# B&R Automation Studio project CombinedLinenSoiledA9KAN
Automation Studio 4.10.2.37

## Configuration CP1584

CPU 5APC2200.AL14-000, AutomationRuntime D4.91, Build 4.1.2, Safety 0.0, Vc V4.72.3

### Task classes (Cpu.sw)
```
Cyclic#2 (cycle 10000 us, tolerance 10000 us):
  zzstd <- Sequences.zzstd.prg
  zztc2str <- Sequences.zztc2str.prg
  zzforcei <- Sequences.zzforcei.prg
  zzconst <- Sequences.zzconst.prg
  zztrip <- Sequences.zztrip.prg
  zzbagsfl <- Sequences.zzbagsfl.prg
  zzbitcal <- Sequences.zzbitcal.prg
  zcusfifo <- Sequences.zcusfifo.prg
  zzStnSer <- Sequences.10ms.zzStnSer.prg
  1_stnsa <- Sequences.10ms.1_stnsa.prg
  2_belt1 <- Sequences.10ms.2_belt1.prg
  3_slu_1 <- Sequences.10ms.3_slu_1.prg
  4_spn1 <- Sequences.10ms.4_spn1.prg
  5_spf1 <- Sequences.10ms.5_spf1.prg
  6_sdc1 <- Sequences.10ms.6_sdc1.prg
  7_sdc2 <- Sequences.10ms.7_sdc2.prg
  8_svc1 <- Sequences.10ms.8_svc1.prg
  9_sic1 <- Sequences.10ms.9_sic1.prg
  10_bson <- Sequences.10ms.10_bson.prg
  11_bsoff <- Sequences.10ms.11_bsoff.prg
  12_svc2 <- Sequences.10ms.12_svc2.prg
  ssr_sortbe <- Sequences.10ms.ssr_sortbelt.prg
  can_live <- Sequences.can_live.prg
  zzio <- Sequences.zzio.prg
  zztcpip <- Sequences.zztcpip.prg
  zzuld_3 <- Sequences.zzuld_3.prg
  zzreport <- Sequences.zzreport.prg
  zztc2end <- Sequences.zztc2end.prg
Cyclic#4:
  Kan_Drv <- Mewa.KanLink.Kan_Drv.prg [disabled]
  mnEth <- Mewa.KGFramework.Pkg_mnEth.mnEth.prg
  BatchInfo <- Mewa.KanLink.BatchInfo.prg
  zzKanLink <- Mewa.KanLink.zzKanLink.prg [disabled]
Cyclic#5:
  zzweigh <- zzweigh.prg
  can_drv2 <- Mewa.200ms.CAN.can_drv2.prg
  zzalarms <- Sequences.zzalarms.prg
  zzstn_q <- Sequences.zzstn_q.prg
  zztime <- zztime.prg
  zztc2end1 <- zztc2end.prg
DataObjects: can_cmd <- Mewa.200ms.CAN.can_cmd.dob
Binaries: TCData, udbdef, sysconf, ashwd, asfw, arconfig, iomap, ashwac, mvLoader
Libraries: DataBackUp, mnParamLib, KanLinkLib, KGstdLib, KL_UserLib, AsDb, standard, runtime, FileIO, Ethernet, dvframe, DataObj, OPERATOR, CAN_Lib, AsTime, AsString, SupLib4, sys_lib, AsTCP, KGstring, Visapi, AsETH, AsBrStr, AsBrWStr, AsUSB, AsMem, AsArLog, AsUDP, brsystem, AsIODiag, AsARCfg, AsIecCon, IecCheck, zzSQL_Lib, arssl
```

### Hardware
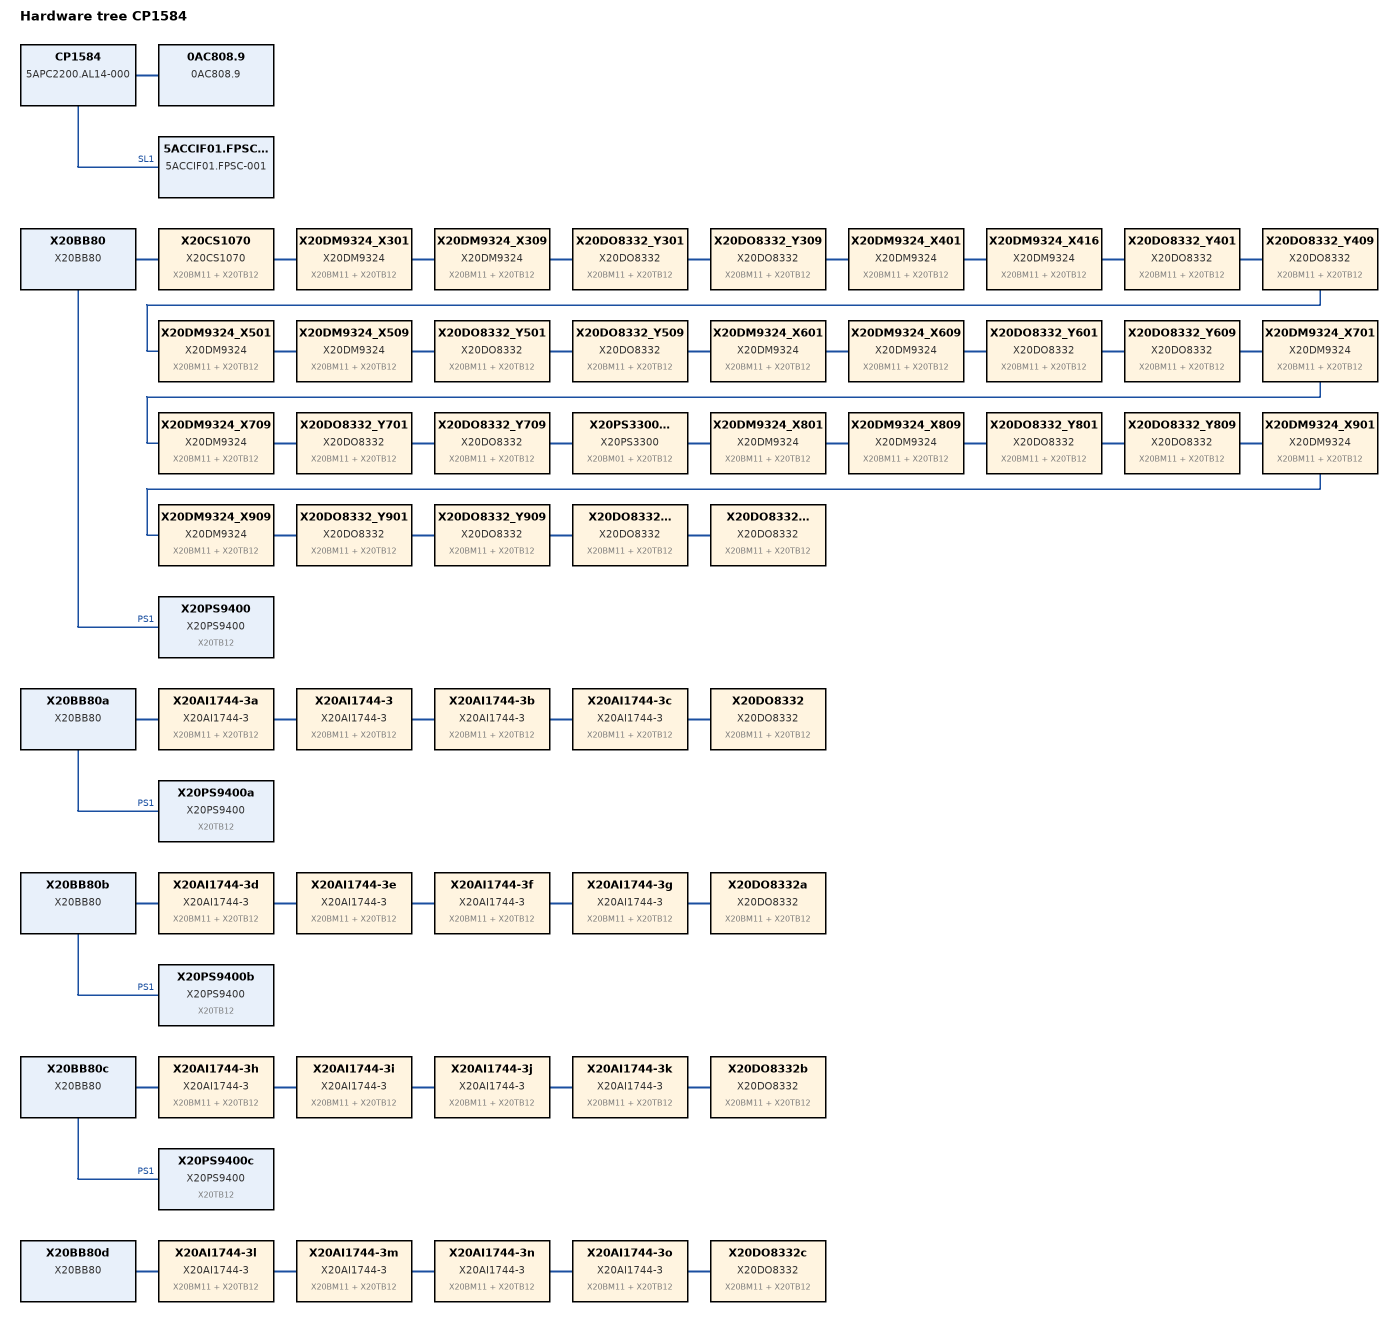
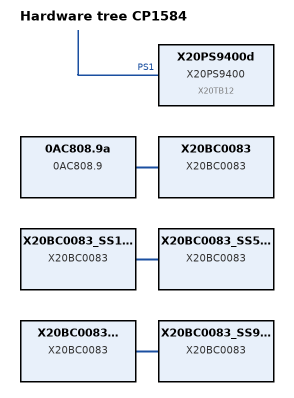
```
0AC808.9 : 0AC808.9 v1.0.0.0  [ETH1 -> CP1584.IF3 [Cable Type=PowerlinkCable, Length=10, Version=1.0.0.3]]
0AC808.9a : 0AC808.9 v1.0.0.0  [ETH2 -> X20BC0083.PLK1 [Cable Type=PowerlinkCable, Length=10, Version=1.0.0.3]; ETH4 -> X20BC0083_SS1-4.PLK2 [Cable Type=PowerlinkCable, Length=10, Version=1.0.0.3]]
5ACCIF01.FPSC-001 : 5ACCIF01.FPSC-001 v1.9.1.0  [SL -> CP1584.SL1]
  Connector IF1:
    DNAConfiguration = manual
CP1584 : 5APC2200.AL14-000 v2.0.3.0
  Connector IF3:
    AssignedOperatingSystem = ARemb
    ActivateDevice = 1
    Baudrate = 100
    InaNodeNumber = 21
    ActivateANSL = 0
  Connector IF4:
    AssignedOperatingSystem = ARemb
    ActivateDevice = 1
    Mode = Manual
    InternetAddress = 10.8.4.20
    SubnetMask = 255.255.240.0
  Connector IF5:
    AssignedOperatingSystem = ARemb
  Connector IF6:
    AssignedOperatingSystem = ARemb
  ConfigurationID = AS4_2_BaseStandard_Supertrack
  UserPartitionSize = 0
  UserRamDevice = PCI.1.PPC21xx.SRAM
  UserRamSize = 200000
  RemMemDevice = PCI.1.PPC21xx.SRAM
  RemMemSize = 200000
  PermanentPvSize = 46756
  RemanentGlobalPvSize = 8944
  VolatileGlobalPvSize = 450000
  EnableUsbRemoteInstall = 1
  EnableCfRemoteInstall = 1
  Cyclic1Duration = 1000
  Cyclic1Tolerance = 1000
  Cyclic2Duration = 10000
  Cyclic2Tolerance = 10000
  FileDevice1
  FileDeviceName1 = USBStick
  FileDevicePath1 = /bd0\
  FileDevice2
  FileDeviceName2 = UserPart
  FileDevicePath2 = F:\
  EthernetHostName = SupertrackPLC
  EthernetDefaultGateway = 10.8.15.254
  FtpUser1
  FtpUsername1 = admin
  FtpUserPassword1 = vwQCGOhDKwuFhUdMhisKVJgiKzmoNTQazzJQnTTJsZU=  // admin
  FtpUserSalt1 = XFuy8Eo/
  FTPAccessRight1 = 0
  ActivateOpcUa = 1
  OpcUaInformationModels_PV_Version = 1
X20AI1744-3 : X20AI1744-3 v1.7.0.0  [SS1 -> X20TB12ai.SS; SL -> X20BM11af.SL1]
  Supervision = off
X20AI1744-3a : X20AI1744-3 v1.7.0.0  [SS1 -> X20TB12ah.SS; SL -> X20BM11ae.SL1]
  Supervision = off
X20AI1744-3b : X20AI1744-3 v1.7.0.0  [SS1 -> X20TB12aj.SS; SL -> X20BM11ag.SL1]
  Supervision = off
X20AI1744-3c : X20AI1744-3 v1.7.0.0  [SS1 -> X20TB12ak.SS; SL -> X20BM11ah.SL1]
  Supervision = off
X20AI1744-3d : X20AI1744-3 v1.7.0.0  [SS1 -> X20TB12ap.SS; SL -> X20BM11aj.SL1]
  Supervision = off
X20AI1744-3e : X20AI1744-3 v1.7.0.0  [SS1 -> X20TB12aq.SS; SL -> X20BM11ak.SL1]
  Supervision = off
X20AI1744-3f : X20AI1744-3 v1.7.0.0  [SS1 -> X20TB12ar.SS; SL -> X20BM11al.SL1]
  Supervision = off
X20AI1744-3g : X20AI1744-3 v1.7.0.0  [SS1 -> X20TB12as.SS; SL -> X20BM11am.SL1]
  Supervision = off
X20AI1744-3h : X20AI1744-3 v1.7.0.0  [SS1 -> X20TB12au.SS; SL -> X20BM11ao.SL1]
  Supervision = off
X20AI1744-3i : X20AI1744-3 v1.7.0.0  [SS1 -> X20TB12av.SS; SL -> X20BM11ap.SL1]
  Supervision = off
X20AI1744-3j : X20AI1744-3 v1.7.0.0  [SS1 -> X20TB12aw.SS; SL -> X20BM11aq.SL1]
  Supervision = off
X20AI1744-3k : X20AI1744-3 v1.7.0.0  [SS1 -> X20TB12ax.SS; SL -> X20BM11ar.SL1]
  Supervision = off
X20AI1744-3l : X20AI1744-3 v1.7.0.0  [SS1 -> X20TB12az.SS; SL -> X20BM11at.SL1]
  Supervision = off
X20AI1744-3m : X20AI1744-3 v1.7.0.0  [SS1 -> X20TB12ba.SS; SL -> X20BM11au.SL1]
  Supervision = off
X20AI1744-3n : X20AI1744-3 v1.7.0.0  [SS1 -> X20TB12bb.SS; SL -> X20BM11av.SL1]
  Supervision = off
X20AI1744-3o : X20AI1744-3 v1.7.0.0  [SS1 -> X20TB12bc.SS; SL -> X20BM11aw.SL1]
  Supervision = off
X20BB80 : X20BB80 v1.1.0.0
X20BB80a : X20BB80 v1.1.0.0
X20BB80b : X20BB80 v1.1.0.0
X20BB80c : X20BB80 v1.1.0.0
X20BB80d : X20BB80 v1.1.0.0
X20BC0083 : X20BC0083 v2.14.0.0  [PLK1 -> 0AC808.9a.ETH2 [Cable Type=PowerlinkCable, Length=10, Version=1.0.0.3]; PLK2 -> 5ACCIF01.FPSC-001.IF1 [Cable Type=PowerlinkCable, Length=10, Version=1.0.0.3]; SL -> X20BB80.SL1]
  Supervision = off
X20BC0083_SS1-4 : X20BC0083 v2.14.0.0  [PLK1 -> X20BC0083_SS5-8.PLK1 [Cable Type=PowerlinkCable, Length=10, Version=1.0.0.3]; PLK2 -> 0AC808.9a.ETH4 [Cable Type=PowerlinkCable, Length=10, Version=1.0.0.3]; SL -> X20BB80a.SL1]
  Supervision = off
X20BC0083_SS13-16 : X20BC0083 v2.14.0.0  [PLK2 -> X20BC0083_SS9-12.PLK1 (NodeNumber=5) [Cable Type=PowerlinkCable, Length=10, Version=1.0.0.3]; SL -> X20BB80d.SL1]
  Supervision = off
X20BC0083_SS5-8 : X20BC0083 v2.14.0.0  [PLK1 -> X20BC0083_SS1-4.PLK1 (NodeNumber=3) [Cable Type=PowerlinkCable, Length=10, Version=1.0.0.3]; PLK2 -> X20BC0083_SS9-12.PLK2 (NodeNumber=3) [Cable Type=PowerlinkCable, Length=10, Version=1.0.0.3]; SL -> X20BB80b.SL1]
  Supervision = off
X20BC0083_SS9-12 : X20BC0083 v2.14.0.0  [PLK1 -> X20BC0083_SS13-16.PLK2 (NodeNumber=4) [Cable Type=PowerlinkCable, Length=10, Version=1.0.0.3]; PLK2 -> X20BC0083_SS5-8.PLK2 (NodeNumber=4) [Cable Type=PowerlinkCable, Length=10, Version=1.0.0.3]; SL -> X20BB80c.SL1]
  Supervision = off
X20BM01 : X20BM01 v2.1.0.0  [X2X1 -> X20BM11t.X2X2]
X20BM11 : X20BM11 v1.1.0.0  [X2X1 -> X20BB80.IF1]
X20BM11a : X20BM11 v1.1.0.0  [X2X1 -> X20BM11.X2X2]
X20BM11aa : X20BM11 v1.1.0.0  [X2X1 -> X20BM11z.X2X2]
X20BM11ab : X20BM11 v1.1.0.0  [X2X1 -> X20BM11aa.X2X2]
X20BM11ac : X20BM11 v1.1.0.0  [X2X1 -> X20BM11ab.X2X2]
X20BM11ad : X20BM11 v1.1.0.0  [X2X1 -> X20BM11ac.X2X2]
X20BM11ae : X20BM11 v1.1.0.0  [X2X1 -> X20BB80a.IF1]
X20BM11af : X20BM11 v1.1.0.0  [X2X1 -> X20BM11ae.X2X2]
X20BM11ag : X20BM11 v1.1.0.0  [X2X1 -> X20BM11af.X2X2]
X20BM11ah : X20BM11 v1.1.0.0  [X2X1 -> X20BM11ag.X2X2]
X20BM11ai : X20BM11 v1.1.0.0  [X2X1 -> X20BM11ah.X2X2]
X20BM11aj : X20BM11 v1.1.0.0  [X2X1 -> X20BB80b.IF1]
X20BM11ak : X20BM11 v1.1.0.0  [X2X1 -> X20BM11aj.X2X2]
X20BM11al : X20BM11 v1.1.0.0  [X2X1 -> X20BM11ak.X2X2]
X20BM11am : X20BM11 v1.1.0.0  [X2X1 -> X20BM11al.X2X2]
X20BM11an : X20BM11 v1.1.0.0  [X2X1 -> X20BM11am.X2X2]
X20BM11ao : X20BM11 v1.1.0.0  [X2X1 -> X20BB80c.IF1]
X20BM11ap : X20BM11 v1.1.0.0  [X2X1 -> X20BM11ao.X2X2]
X20BM11aq : X20BM11 v1.1.0.0  [X2X1 -> X20BM11ap.X2X2]
X20BM11ar : X20BM11 v1.1.0.0  [X2X1 -> X20BM11aq.X2X2]
X20BM11as : X20BM11 v1.1.0.0  [X2X1 -> X20BM11ar.X2X2]
X20BM11at : X20BM11 v1.1.0.0  [X2X1 -> X20BB80d.IF1]
X20BM11au : X20BM11 v1.1.0.0  [X2X1 -> X20BM11at.X2X2]
X20BM11av : X20BM11 v1.1.0.0  [X2X1 -> X20BM11au.X2X2]
X20BM11aw : X20BM11 v1.1.0.0  [X2X1 -> X20BM11av.X2X2]
X20BM11ax : X20BM11 v1.1.0.0  [X2X1 -> X20BM11aw.X2X2]
X20BM11b : X20BM11 v1.1.0.0  [X2X1 -> X20BM11a.X2X2]
X20BM11c : X20BM11 v1.1.0.0  [X2X1 -> X20BM11b.X2X2]
X20BM11d : X20BM11 v1.1.0.0  [X2X1 -> X20BM11e.X2X2]
X20BM11e : X20BM11 v1.1.0.0  [X2X1 -> X20BM11c.X2X2]
X20BM11f : X20BM11 v1.1.0.0  [X2X1 -> X20BM11d.X2X2]
X20BM11g : X20BM11 v1.1.0.0  [X2X1 -> X20BM11s.X2X2]
X20BM11h : X20BM11 v1.1.0.0  [X2X1 -> X20BM11f.X2X2]
X20BM11i : X20BM11 v1.1.0.0  [X2X1 -> X20BM11h.X2X2]
X20BM11j : X20BM11 v1.1.0.0  [X2X1 -> X20BM11i.X2X2]
X20BM11k : X20BM11 v1.1.0.0  [X2X1 -> X20BM11j.X2X2]
X20BM11l : X20BM11 v1.1.0.0  [X2X1 -> X20BM11k.X2X2]
X20BM11m : X20BM11 v1.1.0.0  [X2X1 -> X20BM11l.X2X2]
X20BM11n : X20BM11 v1.1.0.0  [X2X1 -> X20BM11m.X2X2]
X20BM11o : X20BM11 v1.1.0.0  [X2X1 -> X20BM11n.X2X2]
X20BM11p : X20BM11 v1.1.0.0  [X2X1 -> X20BM11o.X2X2]
X20BM11q : X20BM11 v1.1.0.0  [X2X1 -> X20BM11p.X2X2]
X20BM11r : X20BM11 v1.1.0.0  [X2X1 -> X20BM11q.X2X2]
X20BM11s : X20BM11 v1.1.0.0  [X2X1 -> X20BM11r.X2X2]
X20BM11t : X20BM11 v1.1.0.0  [X2X1 -> X20BM11g.X2X2]
X20BM11u : X20BM11 v1.1.0.0  [X2X1 -> X20BM01.X2X2]
X20BM11v : X20BM11 v1.1.0.0  [X2X1 -> X20BM11u.X2X2]
X20BM11w : X20BM11 v1.1.0.0  [X2X1 -> X20BM11v.X2X2]
X20BM11x : X20BM11 v1.1.0.0  [X2X1 -> X20BM11w.X2X2]
X20BM11y : X20BM11 v1.1.0.0  [X2X1 -> X20BM11x.X2X2]
X20BM11z : X20BM11 v1.1.0.0  [X2X1 -> X20BM11y.X2X2]
X20CS1070 : X20CS1070 v1.8.0.0  [SS1 -> X20TB12af.SS; SL -> X20BM11.SL1]
  Connector IF1:
    Baudrate = 250000
  FunctionModel = Stream1xCan
  Supervision = off
X20DM9324_X301 : X20DM9324 v1.2.0.0  [SS1 -> X20TB12a.SS; SL -> X20BM11a.SL1]
  Supervision = off
X20DM9324_X309 : X20DM9324 v1.2.0.0  [SS1 -> X20TB12b.SS; SL -> X20BM11b.SL1]
  Supervision = off
X20DM9324_X401 : X20DM9324 v1.2.0.0  [SS1 -> X20TB12d.SS; SL -> X20BM11d.SL1]
  Supervision = off
X20DM9324_X416 : X20DM9324 v1.2.0.0  [SS1 -> X20TB12f.SS; SL -> X20BM11f.SL1]
  Supervision = off
X20DM9324_X501 : X20DM9324 v1.2.0.0  [SS1 -> X20TB12j.SS; SL -> X20BM11j.SL1]
  Supervision = off
X20DM9324_X509 : X20DM9324 v1.2.0.0  [SS1 -> X20TB12k.SS; SL -> X20BM11k.SL1]
  Supervision = off
X20DM9324_X601 : X20DM9324 v1.2.0.0  [SS1 -> X20TB12n.SS; SL -> X20BM11n.SL1]
  Supervision = off
X20DM9324_X609 : X20DM9324 v1.2.0.0  [SS1 -> X20TB12o.SS; SL -> X20BM11o.SL1]
  Supervision = off
X20DM9324_X701 : X20DM9324 v1.2.0.0  [SS1 -> X20TB12r.SS; SL -> X20BM11r.SL1]
  Supervision = off
X20DM9324_X709 : X20DM9324 v1.2.0.0  [SS1 -> X20TB12s.SS; SL -> X20BM11s.SL1]
  Supervision = off
X20DM9324_X801 : X20DM9324 v1.2.0.0  [SS1 -> X20TB12u.SS; SL -> X20BM11u.SL1]
  Supervision = off
X20DM9324_X809 : X20DM9324 v1.2.0.0  [SS1 -> X20TB12v.SS; SL -> X20BM11v.SL1]
  Supervision = off
X20DM9324_X901 : X20DM9324 v1.2.0.0  [SS1 -> X20TB12z.SS; SL -> X20BM11y.SL1]
  Supervision = off
X20DM9324_X909 : X20DM9324 v1.2.0.0  [SS1 -> X20TB12aa.SS; SL -> X20BM11z.SL1]
  Supervision = off
X20DO8332 : X20DO8332 v1.5.0.0  [SS1 -> X20TB12al.SS; SL -> X20BM11ai.SL1]
  Supervision = off
X20DO8332_Y1001 : X20DO8332 v1.5.0.0  [SS1 -> X20TB12ad.SS; SL -> X20BM11ac.SL1]
  Supervision = off
X20DO8332_Y1009 : X20DO8332 v1.5.0.0  [SS1 -> X20TB12ae.SS; SL -> X20BM11ad.SL1]
  Supervision = off
X20DO8332_Y301 : X20DO8332 v1.5.0.0  [SS1 -> X20TB12c.SS; SL -> X20BM11c.SL1]
  Supervision = off
X20DO8332_Y309 : X20DO8332 v1.5.0.0  [SS1 -> X20TB12e.SS; SL -> X20BM11e.SL1]
  Supervision = off
X20DO8332_Y401 : X20DO8332 v1.5.0.0  [SS1 -> X20TB12h.SS; SL -> X20BM11h.SL1]
  Supervision = off
X20DO8332_Y409 : X20DO8332 v1.5.0.0  [SS1 -> X20TB12i.SS; SL -> X20BM11i.SL1]
  Supervision = off
X20DO8332_Y501 : X20DO8332 v1.5.0.0  [SS1 -> X20TB12l.SS; SL -> X20BM11l.SL1]
  Supervision = off
X20DO8332_Y509 : X20DO8332 v1.5.0.0  [SS1 -> X20TB12m.SS; SL -> X20BM11m.SL1]
  Supervision = off
X20DO8332_Y601 : X20DO8332 v1.5.0.0  [SS1 -> X20TB12p.SS; SL -> X20BM11p.SL1]
  Supervision = off
X20DO8332_Y609 : X20DO8332 v1.5.0.0  [SS1 -> X20TB12q.SS; SL -> X20BM11q.SL1]
  Supervision = off
X20DO8332_Y701 : X20DO8332 v1.5.0.0  [SS1 -> X20TB12g.SS; SL -> X20BM11g.SL1]
  Supervision = off
X20DO8332_Y709 : X20DO8332 v1.5.0.0  [SS1 -> X20TB12t.SS; SL -> X20BM11t.SL1]
  Supervision = off
X20DO8332_Y801 : X20DO8332 v1.5.0.0  [SS1 -> X20TB12x.SS; SL -> X20BM11w.SL1]
  Supervision = off
X20DO8332_Y809 : X20DO8332 v1.5.0.0  [SS1 -> X20TB12y.SS; SL -> X20BM11x.SL1]
  Supervision = off
X20DO8332_Y901 : X20DO8332 v1.5.0.0  [SS1 -> X20TB12ab.SS; SL -> X20BM11aa.SL1]
  Supervision = off
X20DO8332_Y909 : X20DO8332 v1.5.0.0  [SS1 -> X20TB12ac.SS; SL -> X20BM11ab.SL1]
  Supervision = off
X20DO8332a : X20DO8332 v1.5.0.0  [SS1 -> X20TB12at.SS; SL -> X20BM11an.SL1]
  Supervision = off
X20DO8332b : X20DO8332 v1.5.0.0  [SS1 -> X20TB12ay.SS; SL -> X20BM11as.SL1]
  Supervision = off
X20DO8332c : X20DO8332 v1.5.0.0  [SS1 -> X20TB12bd.SS; SL -> X20BM11ax.SL1]
  Supervision = off
X20PS3300_Power : X20PS3300 v1.3.0.0  [SS1 -> X20TB12w.SS; SL -> X20BM01.SL1]
  Supervision = off
X20PS9400 : X20PS9400 v1.8.0.0  [SS1 -> X20TB12.SS; PS -> X20BB80.PS1]
  Supervision = off
X20PS9400a : X20PS9400 v1.8.0.0  [SS1 -> X20TB12ag.SS; PS -> X20BB80a.PS1]
  Supervision = off
X20PS9400b : X20PS9400 v1.8.0.0  [SS1 -> X20TB12am.SS; PS -> X20BB80b.PS1]
  Supervision = off
X20PS9400c : X20PS9400 v1.8.0.0  [SS1 -> X20TB12an.SS; PS -> X20BB80c.PS1]
  Supervision = off
X20PS9400d : X20PS9400 v1.8.0.0  [SS1 -> X20TB12ao.SS; PS -> X20BB80d.PS1]
  Supervision = off
X20TB12 : X20TB12 v1.0.0.0
X20TB12a : X20TB12 v1.0.0.0
X20TB12aa : X20TB12 v1.0.0.0
X20TB12ab : X20TB12 v1.0.0.0
X20TB12ac : X20TB12 v1.0.0.0
X20TB12ad : X20TB12 v1.0.0.0
X20TB12ae : X20TB12 v1.0.0.0
X20TB12af : X20TB12 v1.0.0.0
X20TB12ag : X20TB12 v1.0.0.0
X20TB12ah : X20TB12 v1.0.0.0
X20TB12ai : X20TB12 v1.0.0.0
X20TB12aj : X20TB12 v1.0.0.0
X20TB12ak : X20TB12 v1.0.0.0
X20TB12al : X20TB12 v1.0.0.0
X20TB12am : X20TB12 v1.0.0.0
X20TB12an : X20TB12 v1.0.0.0
X20TB12ao : X20TB12 v1.0.0.0
X20TB12ap : X20TB12 v1.0.0.0
X20TB12aq : X20TB12 v1.0.0.0
X20TB12ar : X20TB12 v1.0.0.0
X20TB12as : X20TB12 v1.0.0.0
X20TB12at : X20TB12 v1.0.0.0
X20TB12au : X20TB12 v1.0.0.0
X20TB12av : X20TB12 v1.0.0.0
X20TB12aw : X20TB12 v1.0.0.0
X20TB12ax : X20TB12 v1.0.0.0
X20TB12ay : X20TB12 v1.0.0.0
X20TB12az : X20TB12 v1.0.0.0
X20TB12b : X20TB12 v1.0.0.0
X20TB12ba : X20TB12 v1.0.0.0
X20TB12bb : X20TB12 v1.0.0.0
X20TB12bc : X20TB12 v1.0.0.0
X20TB12bd : X20TB12 v1.0.0.0
X20TB12c : X20TB12 v1.0.0.0
X20TB12d : X20TB12 v1.0.0.0
X20TB12e : X20TB12 v1.0.0.0
X20TB12f : X20TB12 v1.0.0.0
X20TB12g : X20TB12 v1.0.0.0
X20TB12h : X20TB12 v1.0.0.0
X20TB12i : X20TB12 v1.0.0.0
X20TB12j : X20TB12 v1.0.0.0
X20TB12k : X20TB12 v1.0.0.0
X20TB12l : X20TB12 v1.0.0.0
X20TB12m : X20TB12 v1.0.0.0
X20TB12n : X20TB12 v1.0.0.0
X20TB12o : X20TB12 v1.0.0.0
X20TB12p : X20TB12 v1.0.0.0
X20TB12q : X20TB12 v1.0.0.0
X20TB12r : X20TB12 v1.0.0.0
X20TB12s : X20TB12 v1.0.0.0
X20TB12t : X20TB12 v1.0.0.0
X20TB12u : X20TB12 v1.0.0.0
X20TB12v : X20TB12 v1.0.0.0
X20TB12w : X20TB12 v1.0.0.0
X20TB12x : X20TB12 v1.0.0.0
X20TB12y : X20TB12 v1.0.0.0
X20TB12z : X20TB12 v1.0.0.0
```

### Cpu.per - CP1584/Cpu.per
```iecst
(********************************************************************
 * COPYRIGHT -- HP
 ********************************************************************
 * File: Cpu.per
 * Author: treamsbottom
 * Created: March 03, 2014
 ********************************************************************
 * Declaration of permanent variables
 ********************************************************************)
VAR_CONFIG
	Bag AT %M0; (* *)
	C AT %MW16000; (* *)
	D AT %MW16200; (* *)
	(*D32 AT %MD32200; (* *)
	ReportBuffer AT %M36200; (* *)
	SQL AT %M44200; (* *)
END_VAR
```

### IoMap.iom - CP1584/IoMap.iom
```iecst
(********************************************************************
 * COPYRIGHT --
 ********************************************************************
 * File: IoMap.iom
 * Author: Dave
 * Created: November 19, 2010
 ********************************************************************
 * IO mapping file
 ********************************************************************)
VAR_CONFIG
	X[3].X01 AT %QX."X20DO8332_Y301".DigitalOutput01;
	X[3].X02 AT %QX."X20DO8332_Y301".DigitalOutput02;
	X[3].X03 AT %QX."X20DO8332_Y301".DigitalOutput03;
	X[3].X04 AT %QX."X20DO8332_Y301".DigitalOutput04;
	X[3].X05 AT %QX."X20DO8332_Y301".DigitalOutput05;
	X[3].X06 AT %QX."X20DO8332_Y301".DigitalOutput06;
	X[3].X07 AT %QX."X20DO8332_Y301".DigitalOutput07;
	X[3].X08 AT %QX."X20DO8332_Y301".DigitalOutput08;
	X[3].X09 AT %IX."X20DM9324_X309".DigitalInput01;
	X[3].X10 AT %IX."X20DM9324_X309".DigitalInput02;
	X[3].X11 AT %IX."X20DM9324_X309".DigitalInput03;
	X[3].X12 AT %IX."X20DM9324_X309".DigitalInput04;
	X[3].X13 AT %IX."X20DM9324_X309".DigitalInput05;
	X[3].X14 AT %IX."X20DM9324_X309".DigitalInput06;
	X[3].X15 AT %IX."X20DM9324_X309".DigitalInput07;
	X[3].X16 AT %IX."X20DM9324_X309".DigitalInput08;
	Y[3].Y01 AT %IX."X20DM9324_X301".DigitalInput01;
	Y[3].Y02 AT %IX."X20DM9324_X301".DigitalInput02;
	Y[3].Y03 AT %IX."X20DM9324_X301".DigitalInput03;
	Y[3].Y04 AT %IX."X20DM9324_X301".DigitalInput04;
	Y[3].Y05 AT %IX."X20DM9324_X301".DigitalInput05;
	Y[3].Y06 AT %IX."X20DM9324_X301".DigitalInput06;
	Y[3].Y07 AT %IX."X20DM9324_X301".DigitalInput07;
	Y[3].Y08 AT %IX."X20DM9324_X301".DigitalInput08;
	Y[3].Y09 AT %QX."X20DO8332_Y309".DigitalOutput01;
	Y[3].Y10 AT %QX."X20DO8332_Y309".DigitalOutput02;
	Y[3].Y11 AT %QX."X20DO8332_Y309".DigitalOutput03;
	Y[3].Y12 AT %QX."X20DO8332_Y309".DigitalOutput04;
	Y[3].Y13 AT %QX."X20DO8332_Y309".DigitalOutput05;
	Y[3].Y14 AT %QX."X20DO8332_Y309".DigitalOutput06;
	Y[3].Y15 AT %QX."X20DO8332_Y309".DigitalOutput07;
	Y[3].Y16 AT %QX."X20DO8332_Y309".DigitalOutput08;
	X[4].X01 AT %IX."X20DM9324_X401".DigitalInput01;
	X[4].X02 AT %IX."X20DM9324_X401".DigitalInput02;
	X[4].X03 AT %IX."X20DM9324_X401".DigitalInput03;
	X[4].X04 AT %IX."X20DM9324_X401".DigitalInput04;
	X[4].X05 AT %IX."X20DM9324_X401".DigitalInput05;
	X[4].X06 AT %IX."X20DM9324_X401".DigitalInput06;
	X[4].X07 AT %IX."X20DM9324_X401".DigitalInput07;
	X[4].X08 AT %IX."X20DM9324_X401".DigitalInput08;
	X[4].X09 AT %IX."X20DM9324_X416".DigitalInput01;
	X[4].X10 AT %IX."X20DM9324_X416".DigitalInput02;
	X[4].X11 AT %IX."X20DM9324_X416".DigitalInput03;
	X[4].X12 AT %IX."X20DM9324_X416".DigitalInput04;
	X[4].X13 AT %IX."X20DM9324_X416".DigitalInput05;
	X[4].X14 AT %IX."X20DM9324_X416".DigitalInput06;
	X[4].X15 AT %IX."X20DM9324_X416".DigitalInput07;
	X[4].X16 AT %IX."X20DM9324_X416".DigitalInput08;
	Y[4].Y01 AT %QX."X20DO8332_Y401".DigitalOutput01;
	Y[4].Y02 AT %QX."X20DO8332_Y401".DigitalOutput02;
	Y[4].Y03 AT %QX."X20DO8332_Y401".DigitalOutput03;
	Y[4].Y04 AT %QX."X20DO8332_Y401".DigitalOutput04;
	Y[4].Y05 AT %QX."X20DO8332_Y401".DigitalOutput05;
	Y[4].Y06 AT %QX."X20DO8332_Y401".DigitalOutput06;
	Y[4].Y07 AT %QX."X20DO8332_Y401".DigitalOutput07;
	Y[4].Y08 AT %QX."X20DO8332_Y401".DigitalOutput08;
	Y[4].Y09 AT %QX."X20DO8332_Y409".DigitalOutput01;
	Y[4].Y10 AT %QX."X20DO8332_Y409".DigitalOutput02;
	Y[4].Y11 AT %QX."X20DO8332_Y409".DigitalOutput03;
	Y[4].Y12 AT %QX."X20DO8332_Y409".DigitalOutput04;
	Y[4].Y13 AT %QX."X20DO8332_Y409".DigitalOutput05;
	Y[4].Y14 AT %QX."X20DO8332_Y409".DigitalOutput06;
	Y[4].Y15 AT %QX."X20DO8332_Y409".DigitalOutput07;
	Y[4].Y16 AT %QX."X20DO8332_Y409".DigitalOutput08;
	X[5].X01 AT %IX."X20DM9324_X501".DigitalInput01;
	X[5].X02 AT %IX."X20DM9324_X501".DigitalInput02;
	X[5].X03 AT %IX."X20DM9324_X501".DigitalInput03;
	X[5].X04 AT %IX."X20DM9324_X501".DigitalInput04;
	X[5].X05 AT %IX."X20DM9324_X501".DigitalInput05;
	X[5].X06 AT %IX."X20DM9324_X501".DigitalInput06;
	X[5].X07 AT %IX."X20DM9324_X501".DigitalInput07;
	X[5].X08 AT %IX."X20DM9324_X501".DigitalInput08;
	X[5].X09 AT %IX."X20DM9324_X509".DigitalInput01;
	X[5].X10 AT %IX."X20DM9324_X509".DigitalInput02;
	X[5].X11 AT %IX."X20DM9324_X509".DigitalInput03;
	X[5].X12 AT %IX."X20DM9324_X509".DigitalInput04;
	X[5].X13 AT %IX."X20DM9324_X509".DigitalInput05;
	X[5].X14 AT %IX."X20DM9324_X509".DigitalInput06;
	X[5].X15 AT %IX."X20DM9324_X509".DigitalInput07;
	X[5].X16 AT %IX."X20DM9324_X509".DigitalInput08;
	Y[5].Y01 AT %QX."X20DO8332_Y501".DigitalOutput01;
	Y[5].Y02 AT %QX."X20DO8332_Y501".DigitalOutput02;
	Y[5].Y03 AT %QX."X20DO8332_Y501".DigitalOutput03;
	Y[5].Y04 AT %QX."X20DO8332_Y501".DigitalOutput04;
	Y[5].Y05 AT %QX."X20DO8332_Y501".DigitalOutput05;
	Y[5].Y06 AT %QX."X20DO8332_Y501".DigitalOutput06;
	Y[5].Y07 AT %QX."X20DO8332_Y501".DigitalOutput07;
	Y[5].Y08 AT %QX."X20DO8332_Y501".DigitalOutput08;
	Y[5].Y09 AT %QX."X20DO8332_Y509".DigitalOutput01;
	Y[5].Y10 AT %QX."X20DO8332_Y509".DigitalOutput02;
	Y[5].Y11 AT %QX."X20DO8332_Y509".DigitalOutput03;
	Y[5].Y12 AT %QX."X20DO8332_Y509".DigitalOutput04;
	Y[5].Y13 AT %QX."X20DO8332_Y509".DigitalOutput05;
	Y[5].Y14 AT %QX."X20DO8332_Y509".DigitalOutput06;
	Y[5].Y15 AT %QX."X20DO8332_Y509".DigitalOutput07;
	Y[5].Y16 AT %QX."X20DO8332_Y509".DigitalOutput08;
	X[6].X01 AT %IX."X20DM9324_X601".DigitalInput01;
	X[6].X02 AT %IX."X20DM9324_X601".DigitalInput02;
	X[6].X03 AT %IX."X20DM9324_X601".DigitalInput03;
	X[6].X04 AT %IX."X20DM9324_X601".DigitalInput04;
	X[6].X05 AT %IX."X20DM9324_X601".DigitalInput05;
	X[6].X06 AT %IX."X20DM9324_X601".DigitalInput06;
	X[6].X07 AT %IX."X20DM9324_X601".DigitalInput07;
	X[6].X08 AT %IX."X20DM9324_X601".DigitalInput08;
	X[6].X09 AT %IX."X20DM9324_X609".DigitalInput01;
	X[6].X10 AT %IX."X20DM9324_X609".DigitalInput02;
	X[6].X11 AT %IX."X20DM9324_X609".DigitalInput03;
	X[6].X12 AT %IX."X20DM9324_X609".DigitalInput04;
	X[6].X13 AT %IX."X20DM9324_X609".DigitalInput05;
	X[6].X14 AT %IX."X20DM9324_X609".DigitalInput06;
	X[6].X15 AT %IX."X20DM9324_X609".DigitalInput07;
	X[6].X16 AT %IX."X20DM9324_X609".DigitalInput08;
	Y[6].Y01 AT %QX."X20DO8332_Y601".DigitalOutput01;
	Y[6].Y02 AT %QX."X20DO8332_Y601".DigitalOutput02;
	Y[6].Y03 AT %QX."X20DO8332_Y601".DigitalOutput03;
	Y[6].Y04 AT %QX."X20DO8332_Y601".DigitalOutput04;
	Y[6].Y05 AT %QX."X20DO8332_Y601".DigitalOutput05;
	Y[6].Y06 AT %QX."X20DO8332_Y601".DigitalOutput06;
	Y[6].Y07 AT %QX."X20DO8332_Y601".DigitalOutput07;
	Y[6].Y08 AT %QX."X20DO8332_Y601".DigitalOutput08;
	Y[6].Y09 AT %QX."X20DO8332_Y609".DigitalOutput01;
	Y[6].Y10 AT %QX."X20DO8332_Y609".DigitalOutput02;
	Y[6].Y11 AT %QX."X20DO8332_Y609".DigitalOutput03;
	Y[6].Y12 AT %QX."X20DO8332_Y609".DigitalOutput04;
	Y[6].Y13 AT %QX."X20DO8332_Y609".DigitalOutput05;
	Y[6].Y14 AT %QX."X20DO8332_Y609".DigitalOutput06;
	Y[6].Y15 AT %QX."X20DO8332_Y609".DigitalOutput07;
	Y[6].Y16 AT %QX."X20DO8332_Y609".DigitalOutput08;
	X[7].X01 AT %IX."X20DM9324_X701".DigitalInput01;
	X[7].X02 AT %IX."X20DM9324_X701".DigitalInput02;
	X[7].X03 AT %IX."X20DM9324_X701".DigitalInput03;
	X[7].X04 AT %IX."X20DM9324_X701".DigitalInput04;
	X[7].X05 AT %IX."X20DM9324_X701".DigitalInput05;
	X[7].X06 AT %IX."X20DM9324_X701".DigitalInput06;
	X[7].X07 AT %IX."X20DM9324_X701".DigitalInput07;
	X[7].X08 AT %IX."X20DM9324_X701".DigitalInput08;
	X[7].X09 AT %IX."X20DM9324_X709".DigitalInput01;
	X[7].X10 AT %IX."X20DM9324_X709".DigitalInput02;
	X[7].X11 AT %IX."X20DM9324_X709".DigitalInput03;
	X[7].X12 AT %IX."X20DM9324_X709".DigitalInput04;
	X[7].X13 AT %IX."X20DM9324_X709".DigitalInput05;
	X[7].X14 AT %IX."X20DM9324_X709".DigitalInput06;
	X[7].X15 AT %IX."X20DM9324_X709".DigitalInput07;
	X[7].X16 AT %IX."X20DM9324_X709".DigitalInput08;
	Y[7].Y01 AT %QX."X20DO8332_Y701".DigitalOutput01;
	Y[7].Y02 AT %QX."X20DO8332_Y701".DigitalOutput02;
	Y[7].Y03 AT %QX."X20DO8332_Y701".DigitalOutput03;
	Y[7].Y04 AT %QX."X20DO8332_Y701".DigitalOutput04;
	Y[7].Y05 AT %QX."X20DO8332_Y701".DigitalOutput05;
	Y[7].Y06 AT %QX."X20DO8332_Y701".DigitalOutput06;
	Y[7].Y07 AT %QX."X20DO8332_Y701".DigitalOutput07;
	Y[7].Y08 AT %QX."X20DO8332_Y701".DigitalOutput08;
	Y[7].Y09 AT %QX."X20DO8332_Y709".DigitalOutput01;
	Y[7].Y10 AT %QX."X20DO8332_Y709".DigitalOutput02;
	Y[7].Y11 AT %QX."X20DO8332_Y709".DigitalOutput03;
	Y[7].Y12 AT %QX."X20DO8332_Y709".DigitalOutput04;
	Y[7].Y13 AT %QX."X20DO8332_Y709".DigitalOutput05;
	Y[7].Y14 AT %QX."X20DO8332_Y709".DigitalOutput06;
	Y[7].Y15 AT %QX."X20DO8332_Y709".DigitalOutput07;
	Y[7].Y16 AT %QX."X20DO8332_Y709".DigitalOutput08;
	X[8].X01 AT %IX."X20DM9324_X801".DigitalInput01;
	X[8].X02 AT %IX."X20DM9324_X801".DigitalInput02;
	X[8].X03 AT %IX."X20DM9324_X801".DigitalInput03;
	X[8].X04 AT %IX."X20DM9324_X801".DigitalInput04;
	X[8].X05 AT %IX."X20DM9324_X801".DigitalInput05;
	X[8].X06 AT %IX."X20DM9324_X801".DigitalInput06;
	X[8].X07 AT %IX."X20DM9324_X801".DigitalInput07;
	X[8].X08 AT %IX."X20DM9324_X801".DigitalInput08;
	X[8].X09 AT %IX."X20DM9324_X809".DigitalInput01;
	X[8].X10 AT %IX."X20DM9324_X809".DigitalInput02;
	X[8].X11 AT %IX."X20DM9324_X809".DigitalInput03;
	X[8].X12 AT %IX."X20DM9324_X809".DigitalInput04;
	X[8].X13 AT %IX."X20DM9324_X809".DigitalInput05;
	X[8].X14 AT %IX."X20DM9324_X809".DigitalInput06;
	X[8].X15 AT %IX."X20DM9324_X809".DigitalInput07;
	X[8].X16 AT %IX."X20DM9324_X809".DigitalInput08;
	Y[8].Y01 AT %QX."X20DO8332_Y801".DigitalOutput01;
	Y[8].Y02 AT %QX."X20DO8332_Y801".DigitalOutput02;
	Y[8].Y03 AT %QX."X20DO8332_Y801".DigitalOutput03;
	Y[8].Y04 AT %QX."X20DO8332_Y801".DigitalOutput04;
	Y[8].Y05 AT %QX."X20DO8332_Y801".DigitalOutput05;
	Y[8].Y06 AT %QX."X20DO8332_Y801".DigitalOutput06;
	Y[8].Y07 AT %QX."X20DO8332_Y801".DigitalOutput07;
	Y[8].Y08 AT %QX."X20DO8332_Y801".DigitalOutput08;
	Y[8].Y09 AT %QX."X20DO8332_Y809".DigitalOutput01;
	Y[8].Y10 AT %QX."X20DO8332_Y809".DigitalOutput02;
	Y[8].Y11 AT %QX."X20DO8332_Y809".DigitalOutput03;
	Y[8].Y12 AT %QX."X20DO8332_Y809".DigitalOutput04;
	Y[8].Y13 AT %QX."X20DO8332_Y809".DigitalOutput05;
	Y[8].Y14 AT %QX."X20DO8332_Y809".DigitalOutput06;
	Y[8].Y15 AT %QX."X20DO8332_Y809".DigitalOutput07;
	Y[8].Y16 AT %QX."X20DO8332_Y809".DigitalOutput08;
	X[9].X01 AT %IX."X20DM9324_X901".DigitalInput01;
	X[9].X02 AT %IX."X20DM9324_X901".DigitalInput02;
	X[9].X03 AT %IX."X20DM9324_X901".DigitalInput03;
	X[9].X04 AT %IX."X20DM9324_X901".DigitalInput04;
	X[9].X05 AT %IX."X20DM9324_X901".DigitalInput05;
	X[9].X06 AT %IX."X20DM9324_X901".DigitalInput06;
	X[9].X07 AT %IX."X20DM9324_X901".DigitalInput07;
	X[9].X08 AT %IX."X20DM9324_X901".DigitalInput08;
	X[9].X09 AT %IX."X20DM9324_X909".DigitalInput01;
	X[9].X10 AT %IX."X20DM9324_X909".DigitalInput02;
	X[9].X11 AT %IX."X20DM9324_X909".DigitalInput03;
	X[9].X12 AT %IX."X20DM9324_X909".DigitalInput04;
	X[9].X13 AT %IX."X20DM9324_X909".DigitalInput05;
	X[9].X14 AT %IX."X20DM9324_X909".DigitalInput06;
	X[9].X15 AT %IX."X20DM9324_X909".DigitalInput07;
	X[9].X16 AT %IX."X20DM9324_X909".DigitalInput08;
	Y[9].Y01 AT %QX."X20DO8332_Y901".DigitalOutput01;
	Y[9].Y02 AT %QX."X20DO8332_Y901".DigitalOutput02;
	Y[9].Y03 AT %QX."X20DO8332_Y901".DigitalOutput03;
	Y[9].Y04 AT %QX."X20DO8332_Y901".DigitalOutput04;
	Y[9].Y05 AT %QX."X20DO8332_Y901".DigitalOutput05;
	Y[9].Y06 AT %QX."X20DO8332_Y901".DigitalOutput06;
	Y[9].Y07 AT %QX."X20DO8332_Y901".DigitalOutput07;
	Y[9].Y08 AT %QX."X20DO8332_Y901".DigitalOutput08;
	Y[9].Y09 AT %QX."X20DO8332_Y909".DigitalOutput01;
	Y[9].Y10 AT %QX."X20DO8332_Y909".DigitalOutput02;
	Y[9].Y11 AT %QX."X20DO8332_Y909".DigitalOutput03;
	Y[9].Y12 AT %QX."X20DO8332_Y909".DigitalOutput04;
	Y[9].Y13 AT %QX."X20DO8332_Y909".DigitalOutput05;
	Y[9].Y14 AT %QX."X20DO8332_Y909".DigitalOutput06;
	Y[9].Y15 AT %QX."X20DO8332_Y909".DigitalOutput07;
	Y[9].Y16 AT %QX."X20DO8332_Y909".DigitalOutput08;
	Y[10].Y01 AT %QX."X20DO8332_Y1001".DigitalOutput01;
	Y[10].Y02 AT %QX."X20DO8332_Y1001".DigitalOutput02;
	Y[10].Y03 AT %QX."X20DO8332_Y1001".DigitalOutput03;
	Y[10].Y04 AT %QX."X20DO8332_Y1001".DigitalOutput04;
	Y[10].Y05 AT %QX."X20DO8332_Y1001".DigitalOutput05;
	Y[10].Y06 AT %QX."X20DO8332_Y1001".DigitalOutput06;
	Y[10].Y07 AT %QX."X20DO8332_Y1001".DigitalOutput07;
	Y[10].Y08 AT %QX."X20DO8332_Y1001".DigitalOutput08;
	Y[10].Y09 AT %QX."X20DO8332_Y1009".DigitalOutput01;
	Y[10].Y10 AT %QX."X20DO8332_Y1009".DigitalOutput02;
	Y[10].Y11 AT %QX."X20DO8332_Y1009".DigitalOutput03;
	Y[10].Y12 AT %QX."X20DO8332_Y1009".DigitalOutput04;
	Y[10].Y13 AT %QX."X20DO8332_Y1009".DigitalOutput05;
	Y[10].Y14 AT %QX."X20DO8332_Y1009".DigitalOutput06;
	Y[10].Y15 AT %QX."X20DO8332_Y1009".DigitalOutput07;
	Y[10].Y16 AT %QX."X20DO8332_Y1009".DigitalOutput08;
	AI2744Raw[1] AT %ID."X20AI1744-3a".AnalogInput01;
	AI2744Raw[2] AT %ID."X20AI1744-3".AnalogInput01;
	AI2744Raw[3] AT %ID."X20AI1744-3b".AnalogInput01;
	AI2744Raw[4] AT %ID."X20AI1744-3c".AnalogInput01;
	AI2744Raw[5] AT %ID."X20AI1744-3d".AnalogInput01;
	AI2744Raw[6] AT %ID."X20AI1744-3e".AnalogInput01;
	AI2744Raw[7] AT %ID."X20AI1744-3f".AnalogInput01;
	AI2744Raw[8] AT %ID."X20AI1744-3g".AnalogInput01;
	AI2744Raw[9] AT %ID."X20AI1744-3h".AnalogInput01;
	AI2744Raw[10] AT %ID."X20AI1744-3i".AnalogInput01;
	AI2744Raw[11] AT %ID."X20AI1744-3j".AnalogInput01;
	AI2744Raw[12] AT %ID."X20AI1744-3k".AnalogInput01;
	AI2744Raw[13] AT %ID."X20AI1744-3l".AnalogInput01;
	AI2744Raw[14] AT %ID."X20AI1744-3m".AnalogInput01;
	AI2744Raw[15] AT %ID."X20AI1744-3n".AnalogInput01;
	AI2744Raw[16] AT %ID."X20AI1744-3o".AnalogInput01;
	Y[12].Y01 AT %QX."X20DO8332".DigitalOutput01;
	Y[12].Y02 AT %QX."X20DO8332".DigitalOutput02;
	Y[12].Y03 AT %QX."X20DO8332".DigitalOutput03;
	Y[12].Y04 AT %QX."X20DO8332".DigitalOutput04;
	Y[12].Y05 AT %QX."X20DO8332".DigitalOutput05;
	Y[12].Y06 AT %QX."X20DO8332".DigitalOutput06;
	Y[12].Y07 AT %QX."X20DO8332".DigitalOutput07;
	Y[12].Y08 AT %QX."X20DO8332".DigitalOutput08;
	Y[13].Y01 AT %QX."X20DO8332a".DigitalOutput01;
	Y[13].Y02 AT %QX."X20DO8332a".DigitalOutput02;
	Y[13].Y03 AT %QX."X20DO8332a".DigitalOutput03;
	Y[13].Y04 AT %QX."X20DO8332a".DigitalOutput04;
	Y[13].Y05 AT %QX."X20DO8332a".DigitalOutput05;
	Y[13].Y06 AT %QX."X20DO8332a".DigitalOutput06;
	Y[13].Y07 AT %QX."X20DO8332a".DigitalOutput07;
	Y[13].Y08 AT %QX."X20DO8332a".DigitalOutput08;
	Y[14].Y01 AT %QX."X20DO8332b".DigitalOutput01;
	Y[14].Y02 AT %QX."X20DO8332b".DigitalOutput02;
	Y[14].Y03 AT %QX."X20DO8332b".DigitalOutput03;
	Y[14].Y04 AT %QX."X20DO8332b".DigitalOutput04;
	Y[14].Y05 AT %QX."X20DO8332b".DigitalOutput05;
	Y[14].Y06 AT %QX."X20DO8332b".DigitalOutput06;
	Y[14].Y07 AT %QX."X20DO8332b".DigitalOutput07;
	Y[14].Y08 AT %QX."X20DO8332b".DigitalOutput08;
	Y[15].Y01 AT %QX."X20DO8332c".DigitalOutput01;
	Y[15].Y02 AT %QX."X20DO8332c".DigitalOutput02;
	Y[15].Y03 AT %QX."X20DO8332c".DigitalOutput03;
	Y[15].Y04 AT %QX."X20DO8332c".DigitalOutput04;
	Y[15].Y05 AT %QX."X20DO8332c".DigitalOutput05;
	Y[15].Y06 AT %QX."X20DO8332c".DigitalOutput06;
	Y[15].Y07 AT %QX."X20DO8332c".DigitalOutput07;
	Y[15].Y08 AT %QX."X20DO8332c".DigitalOutput08;
	OK[1] AT %IX."X20BC0083".ModuleOk;
	OK[2] AT %IX."X20BC0083_SS1-4".ModuleOk;
	OK[5]  AT %IX."X20BC0083_SS13-16".ModuleOk;
	OK[4] AT %IX."X20BC0083_SS9-12".ModuleOk;
	OK[3]  AT %IX."X20BC0083_SS5-8".ModuleOk;
END_VAR
```

## Configuration DisplayPCT04

CPU , AutomationRuntime D4.24, Build 4.1.2, Vc V4.24.0

### Task classes (Cpu.sw)
```
Cyclic#4 (cycle 100000 us, tolerance 100000 us):
  zzSQLDrive <- SQL.zzSQLDriver.prg
Binaries: vcrt, vcpk, vcfntttf, verdana, vcctext, arial, verdanab, vccovl, vcpfmtcx, vccbtn, vcdsint, vcpdsw, vcpdpp30, vcshared, vcmgr, vcpfpp30, visvc, vcalarm, vcfile, vccnum, vccstr, vcresman, vcgclass, vcdsloc, arialbd, vcptelo, vctcal, vcchspot, vcbclass, vccline, Data1, vccshape, vcnet, Data102, Data103, vcpdvnc, Data101, arconfig, iomap, asfw, sysconf, ashwd, vccbmp, PCT0403, PCT0401, PCT0402
Libraries: IecCheck, AsString, sys_lib, astcp, visapi, AsDb, dataobj, asarcfg, aseth, fileio, AsIecCon, AsTime, runtime, standard, zzSQL_Lib
```

### Hardware
```
PCT04 : 4PP065.0571-K05 v1.0.2.2
  Connector IF5:
    ActivateDevice = 1
    Mode = Manual
    InternetAddress = 10.8.4.10
    SubnetMask = 255.255.240.0
    Vnc1
    VncVcObjectName1 = PCT04
    VncKeyMappingFile1 = VC\PS2-Keyboard.dis
    VncAuthentication1 = 1
    VncPasswordViewControl1 = medoc
  PermanentPvSize = 17
  RemanentGlobalPvSize = 4300
  VolatileGlobalPvSize = 150000
  Cyclic1Duration = 10000
  Cyclic1Tolerance = 10000
  Cyclic2Duration = 20000
  Cyclic2Tolerance = 20000
  Cyclic3Duration = 50000
  Cyclic3Tolerance = 50000
  Cyclic4Duration = 100000
  Cyclic4Tolerance = 100000
  Cyclic5Duration = 200000
  Cyclic5Tolerance = 200000
  Cyclic6Duration = 500000
  Cyclic6Tolerance = 500000
  Cyclic7Duration = 1000000
  Cyclic7Tolerance = 1000000
  Cyclic8Duration = 10000
  Cyclic8Tolerance = 30000000
  EthernetDefaultGateway = 10.8.15.254
  VcObjectName = PCT04
  KeyMappingFile = 4PP065.0571-K05d.dis
```

## Logical view

Binary libraries used (declarations not repeated): CAN_Lib, KGstring 1.04.0, SupLib4

### Program Logical/Reference/4_ppn1 (IEC) - *ppn

#### ppn.ab
```automation-basic
;--------------------------------------------
;Sequence 0 - XXX0  D[900 + mySeq]
;--------------------------------------------

PROGRAM _INIT
(* init program *)
END_PROGRAM

PROGRAM _CYCLIC

;Inputs
mySeq				= 4	;Sequence number
myIO				= 101
myZone				= 3

I_BagAtSep[1]		= X[myIO].X01
I_BagAtSep[2]		= X[myIO].X02

I_BagInSep[1]	= X[myIO].X03
I_BagInSep[2]	= X[myIO].X04

I_BagReleased	= X[121].X01

myBuffBag[1]		= Line[66].FirstBag
myBuffBag[2]		= Line[65].FirstBag
BufferBag 			= Line[myRelLine].FirstBag

myRelLine			= 90
MaxLines			= 15
MaxBatchSize 		= 3 ; Max number of bags to send from 1 line with out selecting another..

O_SelectLine[1]		= FALSE
O_SelectLine[2]		= FALSE
O_SelectLine[3]		= FALSE

O_OpenSep[1]		= FALSE
O_OpenSep[2]		= FALSE
O_OpenSep[3]		= FALSE

Alarm[mySeq].Name 	= 0
Alarm[mySeq].Bag	= 10000 + mySeq
Alarm[mySeq].Beacon	= TRUE
Alarm[mySeq].Extra	= 0
Alarm[mySeq].Time	= 3000

;Setup Sequence
STEP = D[900 + mySeq]
;Setup Pulse contact
PLS = (STEP <> LASTSTEP)
LASTSTEP = STEP

;Sequence
IF (STEP = 0) THEN
	;Disabled
ENDIF

LOOP n = 1 TO 2 DO
	TON_Settled[n].IN = I_BagAtSep[n]
	TON_Settled[n].PT = 200
	TON_Settled[n] FUB TON_10ms()
	myBag = myBuffBag[n]
	LineValid[n] = TON_Settled[n].Q AND (Bag[myBag].Cat > 0) AND NOT I_BagInSep[n]

	TON_BagInSep[n].IN = I_BagInSep[n]
	TON_BagInSep[n].PT = 200
	TON_BagInSep[n] FUB TON_10ms()
;	;Correct Destination if bags take up more space than data..... Cannot check in search as using 3 BIT's
;	IF LineValid[n] AND (Bag[myBag].Dst > 0) THEN
;		IF Line[Bag[myBag].Dst].Full THEN
;			INC DebugCount
;			Bag[myBag].Dst = 0
;		ENDIF
;	ENDIF
	;Alarms
ENDLOOP
;Step 1 Try to find batch with the same category

TON_10ms((STEP =1),150,ScanUpdate,ScanUpdateET)
IF (STEP = 1) AND ScanUpdate THEN ; Allow short time for trips to settle and first point to change before looking for next batch
	IF (CurrentDest <= 0) OR (CurrentDest > 15) THEN
		CurrentDest = 1
	ENDIF
	IF (CurrentLine <= 0) OR (CurrentLine > 2) THEN
		CurrentLine = 1
	ENDIF
	IF (PrevLine <= 0) OR (PrevLine > 2) THEN
		PrevLine = 1
	ENDIF
	IF (LineBatchCount[CurrentLine] >= MaxBatchSize) AND LineValid[CurrentLine] AND (DestSearchCount > 2) THEN
		LineBatchCount[CurrentLine] = 0
	ENDIF
	myDestLine = Bag[myBuffBag[CurrentLine]].Dst

	IF (myDestLine > 0) AND (myDestLine <= MaxLines) AND Line[myDestLine].Clear AND (D[mySeq] > 0) and NOT Std.HaltSysZone[myZone] THEN
		IF (Bag[BufferBag].Cat = 0) OR ((myDestLine  = PrevDest) AND Line[myRelLine].Clear)  THEN
			CurrentDest = myDestLine
			;Search for line with matching cat starting at the currently selected line. Ensure we do not send more than a certain number of bags from 1 line.
			myBag = myBuffBag[CurrentLine]
			myDestBag	= (Line[myDestLine].LastBag - Line[myDestLine].Space)

			IF LineValid[CurrentLine] AND (LineBatchCount[CurrentLine] < MaxBatchSize) AND NOT I_BagReleased THEN ; Check line is valid
				IF (Bag[myBag].Cat = Bag[myDestBag].Cat) THEN ; Match Cats.
					D[900 + mySeq] = 2
				ELSE IF (Bag[Line[myDestLine].FirstBag].Cat = 0) THEN ; Line is empty
					D[900 + mySeq] = 2
				ELSE IF (DestSearchCount > 2) THEN ; No matches send any bag
					D[900 + mySeq] = 2
				ELSE
					INC CurrentLine ; Search next line.
					INC LineSearchCount
					IF LineSearchCount > 2 THEN ; Search all lines if nothing search next buffer.
						LineSearchCount = 0
						INC DestSearchCount
					ENDIF
				ENDIF
			ELSE
				INC CurrentLine ; Search next line.
				INC LineSearchCount
				IF LineSearchCount > 2 THEN ; Search all lines if nothing search next buffer.
					LineSearchCount = 0
					INC DestSearchCount
				ENDIF
			ENDIF
		ELSE
			INC CurrentLine ; Search next line.
			INC LineSearchCount
			IF LineSearchCount > 2 THEN ; Search all lines if nothing search next buffer.
				LineSearchCount = 0
				INC DestSearchCount
			ENDIF
		ENDIF
;	ELSE IF  (Bag[myBuffBag[CurrentLine]].Cat > 0) THEN
;		Alarm[mySeq].Name = almDestinationNotValid
;		Alarm[mySeq].Time = 0
;		Alarm[mySeq].Bag = myBuffBag[CurrentLine]
	ELSE IF NOT Std.HaltSysZone[myZone] THEN
		IF ((myDestLine > 0) AND (myDestLine <= MaxLines) AND Line[myDestLine].Full AND (D[mySeq] > 0) AND (DestSearchCount > 0)) THEN
			Bag[myBuffBag[CurrentLine]].Dst = 0
			;INC DebugCount
		ENDIF

		INC CurrentLine ; Search next line.
		INC LineSearchCount
		IF LineSearchCount > 2 THEN ; Search all lines if nothing search next buffer.
			LineSearchCount = 0
			INC DestSearchCount
		ENDIF
	ENDIF
ELSE IF (STEP <> 1) THEN
	DestSearchCount = 0
	LineSearchCount	= 0
ENDIF

;Step 2 Select Points if required
TON_10ms(ResetRequired,200,ResetPoints,ResetPointsET)
IF (STEP = 2) THEN
	LOOP n = 1 TO MaxLines DO
		O_SelectDest[n]		= FALSE
	ENDLOOP
	IF (CurrentDest > 0) AND (CurrentDest <= MaxLines )  THEN
		ResetRequired = ((CurrentDest <> PrevDest) OR (CurrentLine <> PrevLine))
		O_SelectDest[CurrentDest] = TRUE
		O_SelectLine[CurrentLine] = TRUE
		IF NOT ResetRequired OR ResetPoints THEN
			;Clear All other line batch Counts
			LOOP n = 1 TO 3 DO
				IF (n <> CurrentLine) THEN
					LineBatchCount[n] = 0
				ENDIF
			ENDLOOP
			D[900 + mySeq] = 3
		ENDIF
	ELSE
		D[900 + mySeq]  = 1 ; Invalid line/Dest selection reset seq
	ENDIF
ENDIF

;Step 3 Release trolley

IF (STEP = 3) THEN
	IF (CurrentDest > 0) AND (CurrentDest <= MaxLines )  THEN
		myDestLine = myRelLine
		myBag = myBuffBag[CurrentLine]
		myDestBag = Line[myRelLine].LastBag
		IF TON_BagInSep[CurrentLine].Q THEN
			Released = TRUE
		ENDIF
		ReleaseValid = (Bag[myBag].Cat > 0) AND Line[myDestLine].Clear
		O_SelectDest[CurrentDest] = TRUE
		O_SelectLine[CurrentLine] = TRUE
		O_OpenSep[CurrentLine] = ReleaseValid AND NOT Released
		IF I_BagReleased THEN
			INC LineBatchCount[CurrentLine]
			PrevDest = CurrentDest
			PrevLine = CurrentLine
			Bag[myDestBag] = Bag[myBag]
			Bag[myBag] = Bag[0]
			D[900 + mySeq] = 1
		ENDIF
		IF (Bag[myBag].Cat = 0)THEN
			Alarm[mySeq].Bag = myBag
			Alarm[mySeq].Name = almBagDataError
		ENDIF
	ELSE
		Alarm[mySeq].Time = 0
		Alarm[mySeq].Name = almGeneralSequence
	ENDIF
ELSE
	Released = FALSE
ENDIF

;ClearBatch Counts

IF ClearCounts THEN
	LOOP n = 1 TO 3 DO
		LineBatchCount[n] = 0
	ENDLOOP
	ClearCounts = FALSE
ENDIF

;Transer Bag Data

LOOP n = 1 TO MaxLines DO

	StorageLineLastBag = Line[n].LastBag
	IF Line[n].Trip AND (Bag[BufferBag].Cat > 0) AND (Bag[BufferBag].Dst = n) AND (Bag[StorageLineLastBag].Cat = 0) THEN

		Bag[StorageLineLastBag] = 	Bag[BufferBag]
		Bag[StorageLineLastBag].Dst = 0
		Bag[BufferBag] = Bag[0]
	ENDIF
	LineSelect[n] = O_SelectDest[n]
	LineReset[n] = NOT O_SelectDest[n] AND (STEP <> 0)
ENDLOOP
;-----------------------------------
;PLC Outputs - adjust to suit system
;-----------------------------------

Y[myIO].Y05 = O_OpenSep[1]
Y[myIO].Y06 = O_OpenSep[2]

Y[myIO].Y07 = O_SelectLine[1]
Y[myIO].Y08 = O_SelectLine[2]

Y[51].Y05 = LineSelect[1]
Y[51].Y07 = LineReset[1]
Y[51].Y06= LineSelect[2]
Y[51].Y08 = LineReset[2]
Y[52].Y05 = LineSelect[3]
Y[52].Y07 = LineReset[3]
Y[52].Y06= LineSelect[4]
Y[52].Y08 = LineReset[4]
Y[53].Y05 = LineSelect[5]
Y[53].Y07 = LineReset[5]
Y[53].Y06= LineSelect[6]
Y[53].Y08 = LineReset[6]
Y[54].Y05 = LineSelect[7]
Y[54].Y07 = LineReset[7]
Y[54].Y06= LineSelect[8]
Y[54].Y08 = LineReset[8]
Y[55].Y05 = LineSelect[9]
Y[55].Y07 = LineReset[9]
Y[55].Y06= LineSelect[10]
Y[55].Y08 = LineReset[10]
Y[56].Y05 = LineSelect[11]
Y[56].Y07 = LineReset[11]
Y[56].Y06= LineSelect[12]
Y[56].Y08 = LineReset[12]

;Alarms
TimerAlarm.IN 		= NOT PLS AND (Alarm[mySeq].Name > 0)
TimerAlarm.PT 		= Alarm[mySeq].Time
TimerAlarm FUB TON_10ms()
Alarm[mySeq].On 	= TimerAlarm.Q
Alarm[mySeq].ET 	= TimerAlarm.ET
Alarm[mySeq].Zone 	= myZone
END_PROGRAM
```

### Program Logical/Reference/5_ppf1 (IEC) - *PPF1 Offgoing lines 1-13

#### ppf.var
```iecst
VAR
	SDC4_Valid : BOOL;
	SDC3_Valid : BOOL;
	ResetPoints : BOOL;
	Released : BOOL;
	SDC5_Valid : BOOL;
	SDC6_Valid : BOOL;
	TestAtStop : BOOL;
	SDC7_Valid : BOOL;
	OffGoingEnable : BOOL;
	IncSettle : BOOL;
	I_BagAtIncline : BOOL;
	TestReleased : BOOL;
	AlarmBagNotProx : BOOL;
	SDC2_Valid : BOOL;
	SDC1_Valid : BOOL;
	O_Reset : BOOL;
	PLS : BOOL;
	RecircValid : BOOL;
	I_InclineBufferStopOpen : BOOL;
	O_Reset3way : BOOL;
	Line14_Valid : BOOL;
	O_SDCBufferOpen : ARRAY[0..4] OF BOOL;
	I_SDCBagAtBuffer : ARRAY[0..4] OF BOOL;
	BufferClear : ARRAY[0..9] OF BOOL;
	O_OpenSep : ARRAY[0..19] OF BOOL;
	I_BagInSep : ARRAY[0..19] OF BOOL;
	O_Select : ARRAY[0..22] OF BOOL;
	LineSelect : ARRAY[0..30] OF BOOL;
	LineSettle : ARRAY[0..30] OF BOOL;
	I_BagAtStop : ARRAY[0..30] OF BOOL;
	LineInList : ARRAY[0..98] OF BOOL;
	ResetPointsET : TIME;
	TimerAlarm : TON_10ms;
	MaxBuffers : UINT;
END_VAR
VAR RETAIN
	FoundLine : UINT;
	Destination : UINT;
END_VAR
VAR
	BestTime : UINT;
END_VAR
VAR RETAIN
	LASTSTEP : UINT;
END_VAR
VAR
	MinLine : UINT;
	STEP : UINT;
	SearchDest : UINT;
	TransitBag : UINT;
	SettleTime : UINT;
	myRelLine : UINT;
	r : UINT;
	mySeq : UINT;
	x : UINT;
	n : UINT;
	MaxLine : UINT;
	LongestSTime : UINT;
	LongestLine : UINT;
	RecircSpaces : UINT;
	BufferBag : ARRAY[0..30] OF UINT;
	BagSettledTime : ARRAY[0..30] OF UINT;
END_VAR
VAR RETAIN
	SelectedBuffer : USINT;
END_VAR
VAR
	myZone : USINT;
	TON_SettledInSep : ARRAY[0..29] OF TON_10ms;
	TestTim : BOOL;
	BagSettledWithDestTime : ARRAY[0..49] OF UINT;
END_VAR
VAR RETAIN
	lineSpeed : ARRAY[0..15] OF linespeed_typ;
END_VAR
VAR
	myStartTime : DATE_AND_TIME;
	myFinishTime : DATE_AND_TIME;
	myTotalTime : LREAL;
	myNumberOfRecords : LREAL;
END_VAR
```

#### ppf.ab
```automation-basic
PROGRAM _CYCLIC

;----------------------------------------
;Sequence 5 - SPF1 Offgoing Points D[900+mySeq]
;----------------------------------------

;Inputs
;------
mySeq		= 5
TransitBag 	= 810
OffGoingEnable 		= ((D[mySeq] > 0) AND NOT Std.HaltSysZone[myZone])
myZone				= 4

myRelLine = 67

I_SDCBagAtBuffer[1] = FALSE;Bag In Discharger
I_SDCBagAtBuffer[2] = FALSE ;Use for single bag buffer
I_SDCBagAtBuffer[3] = FALSE ;X[6].X13 ;Use for single bag buffer
I_SDCBagAtBuffer[4] = FALSE ;X[6].X13 ;Use for single bag buffer

O_SDCBufferOpen[1]  = FALSE ;Use for single bag buffer
O_SDCBufferOpen[2]  = FALSE ;Use for single bag buffer
O_SDCBufferOpen[3]  = FALSE ;Y[6].Y16 ;Use for single bag buffer
O_SDCBufferOpen[4]  = FALSE ;Y[6].Y16 ;Use for single bag buffer

I_BagAtStop[1]	 	= X[71].X01 OR TestAtStop
I_BagAtStop[2] 		= X[72].X01 OR TestAtStop
I_BagAtStop[3] 		= X[73].X01 OR TestAtStop
I_BagAtStop[4] 		= X[74].X01 OR TestAtStop
I_BagAtStop[5] 		= X[75].X01 OR TestAtStop
I_BagAtStop[6] 		= X[76].X01 OR TestAtStop
I_BagAtStop[7] 		= X[77].X01 OR TestAtStop
I_BagAtStop[8] 		= X[78].X01 OR TestAtStop
I_BagAtStop[9] 		= X[79].X01 OR TestAtStop
I_BagAtStop[10] 	= X[80].X01 OR TestAtStop
I_BagAtStop[11] 	= X[81].X01 OR TestAtStop
I_BagAtStop[12] 	= X[82].X01 OR TestAtStop
I_BagAtStop[13] 	= FALSE
I_BagAtStop[14] 	= FALSE
I_BagAtStop[15] 	= X[102].X01 OR TestAtStop

I_BagInSep[1] 	= X[71].X02 OR TestReleased
I_BagInSep[2]	= X[72].X02 OR TestReleased
I_BagInSep[3]	= X[73].X02 OR TestReleased
I_BagInSep[4]	= X[74].X02 OR TestReleased
I_BagInSep[5]	= X[75].X02 OR TestReleased
I_BagInSep[6]	= X[76].X02 OR TestReleased
I_BagInSep[7]	= X[77].X02 OR TestReleased
I_BagInSep[8]	= X[78].X02 OR TestReleased
I_BagInSep[9]	= X[79].X02 OR TestReleased
I_BagInSep[10] 	= X[80].X02 OR TestReleased
I_BagInSep[11] 	= X[81].X02 OR TestReleased
I_BagInSep[12] 	= X[82].X02 OR TestReleased
I_BagInSep[13] 	= FALSE
I_BagInSep[14] 	= FALSE
I_BagInSep[15] 	= X[102].X03 OR TestReleased

O_Reset 			= FALSE
LOOP n = 1 TO 19 DO
	O_OpenSep[n] = FALSE
	TON_SettledInSep[n].IN = I_BagInSep[n]
	TON_SettledInSep[n].PT	= 75
	TON_SettledInSep[n] FUB TON_10ms()

ENDLOOP
;Buffer line configuration
;-------------------------
MaxBuffers			= 1
MinLine				= 1
MaxLine				= 15

LOOP n = 1 TO 6 DO
	BufferClear[n] 		= UnloadingBuffer[n].SpaceBIT > 0
	Uld[n].SDCReady 	= PUP[n].Enabled AND BufferClear[n]
ENDLOOP

Alarm[mySeq].Name 		= 0
Alarm[mySeq].Bag		= TransitBag
Alarm[mySeq].Beacon		= TRUE
Alarm[mySeq].Extra		= 0
Alarm[mySeq].Time		= 45000

;Setup Sequence
;--------------
STEP = D[900 + mySeq]
;Setup Pulse contact
PLS = (STEP <> LASTSTEP)
LASTSTEP = STEP

;Sequence Steps
;--------------
IF (STEP = 0) THEN
	;Disabled
ENDIF

;Step 1 - Reset Points
TON_10ms((STEP = 1),200,ResetPoints,ResetPointsET)
IF (STEP = 1) THEN
	O_Reset 	= TRUE
	FoundLine 	= 0
	Destination = 0
	IF (ResetPoints AND OffGoingEnable) THEN
		D[900+mySeq] = 2
	ENDIF
ENDIF

;Bags on storage line timers
R_TRIG(Std.Clock100ms,IncSettle)
AlarmBagNotProx 	= FALSE
AlarmBagNotProxLine = 0

LOOP n = MinLine TO MaxLine DO

	LineSettle[n]  = (I_BagAtStop[n] AND (Bag[Line[40 + n].FirstBag].Cat > 0)AND NOT I_BagInSep[n] )
	IF IncSettle AND LineSettle[n] THEN
		IF (BagSettledTime[n] <= $FFFF) THEN
			BagSettledTime[n] = BagSettledTime[n] + 1
		ENDIF
		IF (Bag[Line[40 + n].FirstBag].Dst > 0) AND (BagSettledWithDestTime[n] < $FFFF) THEN
			INC BagSettledWithDestTime[n]
		ELSE IF (Bag[Line[40 + n].FirstBag].Dst = 0) THEN
			BagSettledWithDestTime[n] = 0
		ENDIF
	ELSE IF NOT LineSettle[n] THEN
		BagSettledTime[n] = 0
		BagSettledWithDestTime[n] = 0
		;If Bag has destiantion and not at stop then alarm
		IF (Bag[Line[40 + n].FirstBag].Dst > 0) THEN
			Alarm[mySeq].Name	= almBagNotAtProx
			Alarm[mySeq].Bag	= Line[40 + n].FirstBag
			Alarm[mySeq].Extra 	= n
		ELSE IF I_BagInSep[n] THEN
			Alarm[mySeq].Name	= almSwitchFault
			Alarm[mySeq].Bag	= Line[40 + n].FirstBag
			Alarm[mySeq].Extra 	= n
		ENDIF
	ENDIF
	LongestSTime = 0
	LongestTime[n] = 0
ENDLOOP

LOOP n = MinLine TO MaxLine DO
	LineInList[n]  = FALSE
ENDLOOP

;Longest waiting time used for unloading programs..
LOOP n = MinLine TO MaxLine DO
	LongestLine = 0
	LongestSTime = 0
	LOOP x = MinLine TO MaxLine DO
		IF (BagSettledTime[x] > LongestSTime) AND NOT LineInList[x] THEN ;(BagSettledTime[x] > BagSettledTime[n]) AND
			LongestSTime = BagSettledTime[x]
			LongestLine = x
		ENDIF
	ENDLOOP
	LineInList[LongestLine] = TRUE
	LongestTime[n] = LongestLine
ENDLOOP

;Buffer trip not correct alarms
LOOP n = 1 TO MaxBuffers DO
	IF (STEP = 2) AND BufferClear[n] AND NOT Uld[n].SDCReady THEN
		;Alarm[mySeq].Name 	= almSwitchFault - Not direct to buffers
		;Alarm[mySeq].Bag	= BufferBag[n]
	ENDIF
ENDLOOP

;Search for the bag with a valid destination that has been waiting the longest
IF STEP = 2 THEN

	FoundLine 	= 0
	Destination = 0
	BestTime 	= 0
	SettleTime = 15 ;1.5 seconds

	LOOP n = MinLine TO MaxLine DO
		IF ((BagSettledWithDestTime[n] > SettleTime) AND (BagSettledWithDestTime[n] > BestTime)) THEN
			SearchDest = Bag[Line[40 + n].FirstBag].Dst

			SDC1_Valid  = (SearchDest = 21) AND Uld[1].SDCReady
			SDC2_Valid 	= (SearchDest = 22) AND Uld[2].SDCReady
			SDC3_Valid 	= (SearchDest = 23) AND Uld[3].SDCReady
			SDC4_Valid 	= (SearchDest = 24) AND Uld[4].SDCReady
			SDC5_Valid 	= (SearchDest = 25) AND Uld[5].SDCReady
            SDC6_Valid 	= (SearchDest = 26) AND Uld[6].SDCReady
			;SDC7_Valid 	= ((SearchDest = 37) AND Uld[7].SDCReady)
			;RecircValid = ((SearchDest = 30) AND Line[20].Clear AND (Bag[Line[20].LastBag].Cat = 0))
				IF (SDC1_Valid OR SDC2_Valid OR SDC3_Valid OR SDC4_Valid OR SDC5_Valid OR SDC6_Valid) THEN
				FoundLine 	= n
				Destination = SearchDest
				BestTime 	= BagSettledWithDestTime[n]
			ENDIF
		ENDIF
	ENDLOOP

	IF ((FoundLine > 0) AND (Destination > 0) AND OffGoingEnable ) THEN
		IF Line[myRelLine].Clear AND (Bag[TransitBag] .Cat = 0) AND NOT Line[myRelLine].TripFault THEN
			D[900 + mySeq] = 3
		ENDIF
	ENDIF
ENDIF

;Step 3 - Select Line / Open Stop, Until Bag at correct destination
;Clear Line Selections
LOOP n = MinLine TO MaxLine DO
	LineSelect[n] = FALSE
ENDLOOP

IF (STEP = 3) THEN
	LineSelect[FoundLine] = TRUE
	O_OpenSep[FoundLine] = NOT Released
	IF TON_SettledInSep[FoundLine].Q THEN
		Released = TRUE
		myStartTime = CurrentTimestamp
	ENDIF
	IF (Destination >= 21) AND (Destination <= 26) THEN
		Uld[Destination - 20].DischargerStartLine = FoundLine ;Unloading Program
	ENDIF
	IF (Bag[TransitBag] .Cat = 0) AND (Bag[Line[FoundLine + 40].FirstBag].Cat > 0)THEN
		IF PLS THEN
			Bag[TransitBag]  = Bag[Line[FoundLine + 40].FirstBag]
			Bag[Line[FoundLine + 40].FirstBag] 	= Bag[0]
		ENDIF
	ENDIF
	IF Line[myRelLine].Trip THEN
		IF (FoundLine > 0) AND (FoundLine <= MaxLine) THEN
			LOOP x = 99 DOWNTO 1 DO
				lineSpeed[FoundLine].array[x] = lineSpeed[FoundLine].array[x-1]
			ENDLOOP
			myFinishTime = CurrentTimestamp
			lineSpeed[FoundLine].array[0] = UDINT(CurrentTimestamp - myStartTime)/1000
			//Calculate Average Value
			myTotalTime = 0
			LOOP x = 0 TO 99 DO
				IF (lineSpeed[FoundLine].array[x] > 0) THEN
					myTotalTime = myTotalTime + lineSpeed[FoundLine].array[x]
					myNumberOfRecords = x + 1	//allow for 0 based index
				ENDIF
			EXITIF (lineSpeed[FoundLine].array[x] = 0)
			ENDLOOP
			IF (myTotalTime > 0) AND (myNumberOfRecords > 0) THEN
				lineSpeed[FoundLine].avg = (myTotalTime/myNumberOfRecords)
			ENDIF
		ENDIF
		Bag[Line[myRelLine].LastBag] = Bag[TransitBag]
		Bag[TransitBag] = Bag[0]
		D[900 + mySeq] = 1
	ENDIF
	Alarm[mySeq].Name	= almBagNotReleased
ELSE
	Released = FALSE
ENDIF

;Alarms
TimerAlarm.IN = NOT PLS AND (Alarm[mySeq].Name > 0)
TimerAlarm.PT = Alarm[mySeq].Time
TimerAlarm FUB TON_10ms()
Alarm[mySeq].On = TimerAlarm.Q
Alarm[mySeq].ET = TimerAlarm.ET
Alarm[mySeq].Zone 	= myZone
;Outputs
;-------
LOOP n = 1 TO 12 DO
	Y[70 + n].Y03 = O_OpenSep[n]
	Y[70 + n].Y05 = LineSelect[n]
	Y[70 + n].Y07 = O_Reset
ENDLOOP

;Line 15
Y[102].Y05 = O_OpenSep[15]
Y[102].Y07 = LineSelect[15]
Y[102].Y08 = O_Reset

END_PROGRAM
```

#### ppf.typ
```iecst
TYPE
	linespeed_typ : 	STRUCT
		array : ARRAY[0..99]OF UDINT;
		avg : LREAL;
	END_STRUCT;
END_TYPE
```

### Program Logical/Reference/8_pwb3 (IEC) - *PWB3 Weigh beam 3

#### pwb.var
```iecst
VAR RETAIN
	LASTSTEP : UINT;
	PLS : BOOL;
	STEP : UINT;
END_VAR
VAR
	TimerAlarm : TON_10ms;
	mySeq : UINT;
	myIO : UINT;
	myBag : UINT;
	myRelLine : UINT;
	I_BagInBeam : BOOL;
	O_OpenSep : BOOL;
	myLP : UINT;
	WeighBeamClear : BOOL;
	SettleTime : UDINT;
	BagSettled : BOOL;
	BagSettledET : UDINT;
	RawWgt : DINT;
	Wgt : INT;
	OkToRelease : BOOL;
	myOutBag : UINT;
	myDisplayBag : UINT;
	myZone : INT;
END_VAR
```

### Program Logical/Reference/9_pup1 (IEC) - *PUP1 Unloading point

#### pup.var
```iecst
VAR RETAIN
	LASTSTEP : UINT;
	PLS : BOOL;
	STEP : UINT;
END_VAR
VAR
	TimerAlarm : TON_10ms;
	mySeq : UINT;
	myIO : UINT;
	I_ReleasePB : BOOL;
	I_UnloadingPointOn : BOOL;
	I_TrolleyReleased : BOOL;
	I_BagAtBuffer : BOOL;
	I_BagReleasedBuffer : BOOL;
	myBag : UINT;
	O_Lamp : BOOL;
	O_OpenBuffer : BOOL;
	O_Release : BOOL;
	myPup : UINT;
	SettledBuffer : BOOL;
	SettledBufferET : UDINT;
	myBufferBag : UINT;
	BagReleased : BOOL;
	myZone : INT;
	I_BagInSep : BOOL;
	SettledInSep : BOOL;
	SettledInSepET : UDINT;
END_VAR
```

#### pup.ab
```automation-basic
;--------------------------------------------
;Sequence 0 - XXX0  D[900 + mySeq]
;--------------------------------------------

PROGRAM _INIT
(* init program *)
END_PROGRAM

PROGRAM _CYCLIC

;Inputs
mySeq				= 9	;Sequence number
myIO				= 345
myBufferBag			= 950
myBag				= 987
myPup				= 1
myZone				= 0

I_BagAtBuffer		= X[myIO].X01
I_BagInSep			= X[myIO].X02
I_UnloadingPointOn	= X[myIO].X03
I_ReleasePB			= X[myIO].X04
I_TrolleyReleased	= X[myIO].X08 ; Also Line full

;O_Lamp				= FALSE
PUP[myPup].WorkingLamp = FALSE
O_OpenBuffer		= FALSE
O_Release			= FALSE

Alarm[mySeq].Name 	= 0
Alarm[mySeq].Bag	= myBag
Alarm[mySeq].Beacon	= TRUE
Alarm[mySeq].Extra	= 0
Alarm[mySeq].Time	= 3000

PUP[myPup].Enabled = (D[mySeq] > 0) AND I_UnloadingPointOn ;AND NOT Std.HaltSysZone[myZone]

IF PUP[myPup].Enabled THEN
	PUP[myPup].WorkingLamp = TRUE ; Lamp will display the Unloading point is turned on and flash when off but bags still in transit
ELSE IF (UnloadingBuffer[myPup].CountBIT > 0) THEN
	PUP[myPup].WorkingLamp = Std.Clock1s
ENDIF
O_Lamp = PUP[myPup].WorkingLamp

;Setup Sequence
STEP = D[900 + mySeq]
;Setup Pulse contact
PLS = (STEP <> LASTSTEP)
LASTSTEP = STEP

;Sequence
IF (STEP = 0) THEN
	;Disabled
ENDIF

;Step 1 Wiat for bag at buffer.
TON_10ms(I_BagAtBuffer,75,SettledBuffer,SettledBufferET)
IF (STEP = 1) THEN
	IF (PUP[myPup].Enabled AND SettledBuffer AND (Bag[myBufferBag].Cat > 0) AND (Bag[myBag].Cat = 0) AND NOT I_BagInSep AND NOT Std.HaltSysZone[myZone]) THEN
		D[900 + mySeq] = 2
	ELSE IF I_BagInSep THEN
		Alarm[mySeq].Bag = myBufferBag
		Alarm[mySeq].Name = almSwitchFault
	ELSE IF SettledBuffer AND (Bag[myBufferBag].Cat = 0) THEN
		Alarm[mySeq].Bag = myBufferBag
		Alarm[mySeq].Name = almSwitchFault
	ELSE IF (Bag[myBag].Cat > 0) THEN
		Alarm[mySeq].Name = almBagDataError
	ENDIF
ENDIF

;Step 2 Release bag from Buffer
TON_10ms(I_BagInSep,150,SettledInSep,SettledInSepET)
IF (STEP = 2) THEN
	O_OpenBuffer = NOT SettledInSep
	IF SettledInSep AND (Bag[myBufferBag].Cat > 0) AND (Bag[myBag].Cat = 0) THEN
		Bag[myBag] = Bag[myBufferBag]
		Bag[myBufferBag] = Bag[0]
		D[900 + mySeq] = 3
	ENDIF
	IF (Bag[myBufferBag].Cat = 0) THEN
		Alarm[mySeq].Bag = myBufferBag
		Alarm[mySeq].Name = almBagDataError
	ELSE IF (Bag[myBag].Cat > 0) THEN
		Alarm[mySeq].Name = almBagDataError
	ELSE
		Alarm[mySeq].Bag = myBufferBag
		Alarm[mySeq].Name = almBagNotReleased
	ENDIF
ENDIF

;Step 3 wait for pushbutton to request release of trolley
IF (STEP = 3) THEN
	IF I_ReleasePB AND (ReportUnloading[myPup].Cat = 0) THEN
		ReportUnloading[myPup].Prg = Bag[myBag].Prg 		;Program
		ReportUnloading[myPup].Cat = Bag[myBag].Cat		;Category
		ReportUnloading[myPup].Cus = Bag[myBag].Cus		;Customer
		ReportUnloading[myPup].Wgt = Bag[myBag].Wgt		;Weight
		ReportUnloading[myPup].Cnt = 0					;Count
		ReportUnloading[myPup].Stn = 0					;Station
		ReportUnloading[myPup].Mcn = myPup				;Machine
		ReportUnloading[myPup].Mis = Bag[myBag].Mis		;Batch ID

		Bag[myBag].Cat = Std.MaxCats
		Bag[myBag].Prg = Std.MaxProg
		Bag[myBag].Cus = Std.MaxCust
		D[900 + mySeq] = 4
	ELSE IF (ReportUnloading[myPup].Cat > 0) THEN
		Alarm[mySeq].Name = almGeneralSequence
	ENDIF
ENDIF

;STEP 4 Check for space in empty trolley buffer.
IF (STEP = 4) THEN
	IF NOT I_TrolleyReleased AND NOT Std.HaltSysZone[myZone] THEN
		D[900 + mySeq] = 5
	ENDIF
ENDIF

;STEP 5 Release trolley
IF (STEP = 5) THEN
	O_Release = TRUE
	IF 	I_TrolleyReleased THEN
		Bag[myBag] = Bag[0]
		D[900 + mySeq] = 1
	ENDIF
	Alarm[mySeq].Name = almBagNotReleased
ENDIF

;-----------------------------------
;PLC Outputs - adjust to suit system
;-----------------------------------

Y[myIO].Y05 = O_OpenBuffer
Y[myIO].Y06 = O_Release
Y[myIO].Y07 = O_Lamp

;Alarms
TimerAlarm.IN 		= NOT PLS AND (Alarm[mySeq].Name > 0)
TimerAlarm.PT 		= Alarm[mySeq].Time
TimerAlarm FUB TON_10ms()
Alarm[mySeq].On 	= TimerAlarm.Q
Alarm[mySeq].ET 	= TimerAlarm.ET
Alarm[mySeq].Zone 	= myZone
END_PROGRAM
```

### Program Logical/Reference/12_pup4 (IEC) - *PUP4 Unloading point

#### pup.var
```iecst
VAR RETAIN
	LASTSTEP : UINT;
	PLS : BOOL;
	STEP : UINT;
END_VAR
VAR
	TimerAlarm : TON_10ms;
	mySeq : UINT;
	myIO : UINT;
	I_ReleasePB : BOOL;
	I_UnloadingPointOn : BOOL;
	I_TrolleyReleased : BOOL;
	I_BagAtBuffer : BOOL;
	I_BagReleasedBuffer : BOOL;
	myBag : UINT;
	O_Lamp : BOOL;
	O_OpenBuffer : BOOL;
	O_Release : BOOL;
	myPup : UINT;
	SettledBuffer : BOOL;
	SettledBufferET : UDINT;
	myBufferBag : UINT;
	myZone : INT;
	I_BagInSep : BOOL;
	SettledInSep : BOOL;
	SettledInSepET : UDINT;
END_VAR
```

#### pup.ab
```automation-basic
;--------------------------------------------
;Sequence 0 - XXX0  D[900 + mySeq]
;--------------------------------------------

PROGRAM _INIT
(* init program *)
END_PROGRAM

PROGRAM _CYCLIC

;Inputs
mySeq				= 12	;Sequence number
myIO				= 348
myBufferBag			= 945
myBag				= 997
myPup				= 4
myZone	= 0

I_BagAtBuffer		= X[myIO].X01
I_BagInSep			= X[myIO].X02
I_UnloadingPointOn	= X[myIO].X03
I_ReleasePB			= X[myIO].X04
I_TrolleyReleased	= X[myIO].X08 ; Also Line full

;O_Lamp				= FALSE
PUP[myPup].WorkingLamp = FALSE
O_OpenBuffer		= FALSE
O_Release			= FALSE

Alarm[mySeq].Name 	= 0
Alarm[mySeq].Bag	= myBag
Alarm[mySeq].Beacon	= TRUE
Alarm[mySeq].Extra	= 0
Alarm[mySeq].Time	= 3000

PUP[myPup].Enabled = (D[mySeq] > 0) AND I_UnloadingPointOn

IF PUP[myPup].Enabled THEN
	PUP[myPup].WorkingLamp = TRUE ; Lamp will display the Unloading point is turned on and flash when off but bags still in transit
ELSE IF (UnloadingBuffer[myPup].CountBIT > 0) THEN
	PUP[myPup].WorkingLamp = Std.Clock1s
ENDIF
O_Lamp = PUP[myPup].WorkingLamp

;Setup Sequence
STEP = D[900 + mySeq]
;Setup Pulse contact
PLS = (STEP <> LASTSTEP)
LASTSTEP = STEP

;Sequence
IF (STEP = 0) THEN
	;Disabled
ENDIF

;Step 1 Wiat for bag at buffer.
TON_10ms(I_BagAtBuffer,75,SettledBuffer,SettledBufferET)
IF (STEP = 1) THEN
	IF (PUP[myPup].Enabled AND SettledBuffer AND (Bag[myBufferBag].Cat > 0) AND (Bag[myBag].Cat = 0) AND NOT I_BagInSep AND NOT Std.HaltSysZone[myZone]) THEN
		D[900 + mySeq] = 2
	ELSE IF I_BagInSep THEN
		Alarm[mySeq].Bag = myBufferBag
		Alarm[mySeq].Name = almSwitchFault
	ELSE IF SettledBuffer AND (Bag[myBufferBag].Cat = 0) THEN
		Alarm[mySeq].Bag = myBufferBag
		Alarm[mySeq].Name = almSwitchFault
	ELSE IF (Bag[myBag].Cat > 0) THEN
		Alarm[mySeq].Name = almBagDataError
	ENDIF
ENDIF

;Step 2 Release bag from Buffer
TON_10ms(I_BagInSep,150,SettledInSep,SettledInSepET)
IF (STEP = 2) THEN
	O_OpenBuffer = NOT SettledInSep
	IF SettledInSep AND (Bag[myBufferBag].Cat > 0) AND (Bag[myBag].Cat = 0) THEN
		Bag[myBag] = Bag[myBufferBag]
		Bag[myBufferBag] = Bag[0]
		D[900 + mySeq] = 3
	ENDIF
	IF (Bag[myBufferBag].Cat = 0) THEN
		Alarm[mySeq].Bag = myBufferBag
		Alarm[mySeq].Name = almBagDataError
	ELSE IF (Bag[myBag].Cat > 0) THEN
		Alarm[mySeq].Name = almBagDataError
	ELSE
		Alarm[mySeq].Bag = myBufferBag
		Alarm[mySeq].Name = almBagNotReleased
	ENDIF
ENDIF

;Step 3 wait for pushbutton to request release of trolley
IF (STEP = 3) THEN
	IF I_ReleasePB AND (ReportUnloading[myPup].Cat = 0) THEN
		ReportUnloading[myPup].Prg = Bag[myBag].Prg 		;Program
		ReportUnloading[myPup].Cat = Bag[myBag].Cat		;Category
		ReportUnloading[myPup].Cus = Bag[myBag].Cus		;Customer
		ReportUnloading[myPup].Wgt = Bag[myBag].Wgt		;Weight
		ReportUnloading[myPup].Cnt = 0					;Count
		ReportUnloading[myPup].Stn = 0					;Station
		ReportUnloading[myPup].Mcn = myPup				;Machine
		ReportUnloading[myPup].Mis = Bag[myBag].Mis		;Batch ID

		Bag[myBag].Cat = Std.MaxCats
		Bag[myBag].Prg = Std.MaxProg
		Bag[myBag].Cus = Std.MaxCust
		D[900 + mySeq] = 4
	ELSE IF (ReportUnloading[myPup].Cat > 0) THEN
		Alarm[mySeq].Name = almGeneralSequence
	ENDIF
ENDIF

;STEP 4 Check for space in empty trolley buffer.
IF (STEP = 4) THEN
	IF NOT I_TrolleyReleased AND NOT Std.HaltSysZone[myZone] THEN
		D[900 + mySeq] = 5
	ENDIF
ENDIF

;STEP 5 Release trolley
IF (STEP = 5) THEN
	O_Release = TRUE
	IF 	I_TrolleyReleased THEN
		Bag[myBag] = Bag[0]
		D[900 + mySeq] = 1
	ENDIF
	Alarm[mySeq].Name = almBagNotReleased
ENDIF

;-----------------------------------
;PLC Outputs - adjust to suit system
;-----------------------------------

Y[myIO].Y05 = O_OpenBuffer
Y[myIO].Y06 = O_Release
Y[myIO].Y07 = O_Lamp

;Alarms
TimerAlarm.IN 		= NOT PLS AND (Alarm[mySeq].Name > 0)
TimerAlarm.PT 		= Alarm[mySeq].Time
TimerAlarm FUB TON_10ms()
Alarm[mySeq].On 	= TimerAlarm.Q
Alarm[mySeq].ET 	= TimerAlarm.ET
Alarm[mySeq].Zone 	= myZone
END_PROGRAM
```

### Program Logical/Reference/13_pup5 (IEC) - *PUP5 Unloading point

#### pup.ab
```automation-basic
;--------------------------------------------
;Sequence 0 - XXX0  D[900 + mySeq]
;--------------------------------------------

PROGRAM _INIT
(* init program *)
END_PROGRAM

PROGRAM _CYCLIC

;Inputs
mySeq				= 13	;Sequence number
myIO				= 349
myBag				= 998
myPup				= 5
myZone	= 0

I_UnloadingPointOn	= X[myIO].X03
I_ReleasePB			= X[myIO].X04
I_TrolleyReleased	= X[myIO].X08 ; Also Line full

;O_Lamp				= FALSE
PUP[myPup].WorkingLamp = FALSE
O_OpenBuffer		= FALSE
O_Release			= FALSE
Request.UP[myPup]	= FALSE

Alarm[mySeq].Name 	= 0
Alarm[mySeq].Bag	= myBag
Alarm[mySeq].Beacon	= TRUE
Alarm[mySeq].Extra	= 0
Alarm[mySeq].Time	= 3000

PUP[myPup].Enabled = (D[mySeq] > 0) AND I_UnloadingPointOn

IF PUP[myPup].Enabled THEN
	PUP[myPup].WorkingLamp = TRUE ; Lamp will display the Unloading point is turned on and flash when off but bags still in transit
ELSE IF (UnloadingBuffer[myPup].CountBIT > 0) THEN
	PUP[myPup].WorkingLamp = Std.Clock1s
ENDIF
O_Lamp = PUP[myPup].WorkingLamp

;Setup Sequence
STEP = D[900 + mySeq]
;Setup Pulse contact
PLS = (STEP <> LASTSTEP)
LASTSTEP = STEP

;Sequence
IF (STEP = 0) THEN
	;Disabled
ENDIF

;Step 1 Request a bag from PP
IF (STEP = 1) THEN
	PUPValid = (PUP[myPup].Enabled AND (Bag[myBag].Cat = 0) AND NOT Std.HaltSysZone[myZone])
	Request.UP[myPup] = PUPValid
	IF (Bag[myBag].Cat > 0) AND NOT I_ReleasePB THEN
		D[900 + mySeq] = 2
	ENDIF
ENDIF

;Step 2 wait for pushbutton to request release of trolley
IF (STEP = 2) THEN
	IF I_ReleasePB AND (ReportUnloading[myPup].Cat = 0) THEN
		ReportUnloading[myPup].Prg = Bag[myBag].Prg 		;Program
		ReportUnloading[myPup].Cat = Bag[myBag].Cat		;Category
		ReportUnloading[myPup].Cus = Bag[myBag].Cus		;Customer
		ReportUnloading[myPup].Wgt = Bag[myBag].Wgt		;Weight
		ReportUnloading[myPup].Cnt = 0					;Count
		ReportUnloading[myPup].Stn = 0					;Station
		ReportUnloading[myPup].Mcn = myPup				;Machine
		ReportUnloading[myPup].Mis = Bag[myBag].Mis		;Batch ID

		Bag[myBag].Cat = Std.MaxCats
		Bag[myBag].Prg = Std.MaxProg
		Bag[myBag].Cus = Std.MaxCust
		D[900 + mySeq] = 3
	ELSE IF (ReportUnloading[myPup].Cat > 0) THEN
		Alarm[mySeq].Name = almGeneralSequence
	ENDIF
ENDIF

;STEP 3 Check for space in empty trolley buffer.
IF (STEP = 3) THEN
	IF NOT I_TrolleyReleased AND NOT Std.HaltSysZone[myZone] THEN
		D[900 + mySeq] = 4
	ENDIF
ENDIF

;STEP 4 Release trolley
IF (STEP = 4) THEN
	O_Release = TRUE
	IF 	I_TrolleyReleased THEN
		Bag[myBag] = Bag[0]
		D[900 + mySeq] = 1
	ENDIF
	Alarm[mySeq].Name = almBagNotReleased
ENDIF

;-----------------------------------
;PLC Outputs - adjust to suit system
;-----------------------------------

Y[myIO].Y06 = O_Release
Y[myIO].Y07 = O_Lamp

;Alarms
TimerAlarm.IN 		= NOT PLS AND (Alarm[mySeq].Name > 0)
TimerAlarm.PT 		= Alarm[mySeq].Time
TimerAlarm FUB TON_10ms()
Alarm[mySeq].On 	= TimerAlarm.Q
Alarm[mySeq].ET 	= TimerAlarm.ET
Alarm[mySeq].Zone 	= myZone
END_PROGRAM
```

### Program Logical/Reference/15_pbr1 (IEC) - *PBR1 Bag Remover

#### pbr.var
```iecst
VAR
	LocatedET : TIME;
	Settled : BOOL;
	SettledET : TIME;
	Step3TimedOutET : TIME;
	Step3TimedOut : BOOL;
	SettledAtRemoverET : TIME;
	SettledAtRemover : BOOL;
	STEP : UINT;
	PLS : BOOL;
	LASTSTEP : UINT;
	SeparatorOpened : BOOL;
	SeparatorOpenedET : TIME;
	zzTON_10ms00000 : TON_10ms;
	O_OpenStop : BOOL;
	zzTON_10ms00001 : TON_10ms;
	O_Locate : BOOL;
	O_OpenSeparator : BOOL;
	I_BagReleased : BOOL;
	I_BagAtRemover : BOOL;
	I_BagAtSeparator : BOOL;
	zzTON_10ms00002 : TON_10ms;
	Located : BOOL;
	Step6TimedOutET : TIME;
	Step6TimedOut : BOOL;
	zzTON_10ms00003 : TON_10ms;
	zzTON_10ms00004 : TON_10ms;
	zzTON_10ms00005 : TON_10ms;
	RemoveLocateET : TIME;
	RemoveLocate : BOOL;
	zzTON_10ms00006 : TON_10ms;
	mySeq : UINT;
	TimerAlarm : TON_10ms;
	myIO : UINT;
	myPbr : UINT;
	myZone : UINT;
END_VAR
```

#### pbr.ab
```automation-basic
PROGRAM _INIT
	(* init program *)
END_PROGRAM

PROGRAM _CYCLIC
	(* cyclic program *)

;Sequence 1- Primary Bag remover 1 D[900 + mySeq]

;-----------------------------------------
;Revision 1.00 12/11/2002 D.J. First Issue
;-----------------------------------------
mySeq   = 15
myIO	= 251
myPbr	= 1
myZone	= 0

I_BagAtSeparator	= X[myIO].X01
I_BagAtRemover		= X[myIO].X02
I_BagReleased		= X[myIO].X03

O_OpenSeparator		= FALSE
O_Locate			= FALSE
O_OpenStop			= FALSE

;Setup Sequence
;-----------------------
STEP = D[900 + mySeq]
;Setup Pulse contact
PLS = (STEP <> LASTSTEP)
LASTSTEP = STEP

;Alarm
Alarm[mySeq].Name 	= 0
Alarm[mySeq].Bag	= 0
Alarm[mySeq].Beacon	= TRUE
Alarm[mySeq].Extra	= 0
Alarm[mySeq].Time	= 3000

;Sequence
IF (STEP = 0) THEN
;Disabled
ENDIF

;Wait for bag at separator
IF (STEP = 1) THEN
	O_OpenSeparator = TRUE
	IF I_BagAtRemover THEN
		D[900 + mySeq] = 3
	ELSE IF I_BagAtSeparator THEN
		D[900 + mySeq] = 2
	ENDIF
ENDIF

;Open separator
;Was 3 seconds
TON_10ms((STEP = 2),50,SeparatorOpened,SeparatorOpenedET)
IF (STEP = 2) THEN
	;O_OpenSeparator = TRUE
	IF SeparatorOpened THEN
		D[900 + mySeq] = 3
	ENDIF
ENDIF

;Wait for bag at remover
;Was 3.5 Seconds
TON_10ms(I_BagAtRemover,200,SettledAtRemover,SettledAtRemoverET)
TON_10ms((STEP = 3),2000,Step3TimedOut,Step3TimedOutET)
IF (STEP = 3) THEN
	;O_OpenSeparator = TRUE
	IF SettledAtRemover THEN;AND NOT I_BagReleased) THEN
		D[900 + mySeq] = 4
	ELSE IF Step3TimedOut THEN; AND NOT I_BagReleased) THEN
		D[900 + mySeq] = 1
	ENDIF
ENDIF

;Allow bag to settle
;Was 4 seconds
TON_10ms((STEP = 4),200,Settled,SettledET)
IF (STEP = 4) THEN
	IF (CAN[1].OkToRelease[myPbr] AND Settled AND NOT I_BagReleased) THEN ;(Settled OR I_BagReleased)) THEN
		D[900 + mySeq] = 5
	ENDIF
ENDIF

;Locate hook
;Was 5 seconds
TON_10ms((STEP = 5),300,Located,LocatedET)
IF (STEP = 5) THEN
	O_Locate = TRUE
	IF Located OR I_BagReleased THEN
		D[900 + mySeq] = 6
	ENDIF
ENDIF

;Strip bag
TON_10ms((STEP = 6),1000,Step6TimedOut,Step6TimedOutET)
TON_10ms((STEP = 6),200,RemoveLocate,RemoveLocateET)
IF (STEP = 6) THEN
	O_Locate 	= NOT RemoveLocate
	O_OpenStop 	= TRUE
	IF I_BagReleased THEN
		D[900 + mySeq] = 1
	ELSE IF Step6TimedOut THEN
		D[900 + mySeq] = 4
	ENDIF
ENDIF

;Alarms
TimerAlarm.IN 		= NOT PLS AND (Alarm[mySeq].Name > 0)
TimerAlarm.PT 		= Alarm[mySeq].Time
TimerAlarm FUB TON_10ms()
Alarm[mySeq].On 	= TimerAlarm.Q
Alarm[mySeq].ET 	= TimerAlarm.ET
Alarm[mySeq].Zone 	= myZone

Y[myIO].Y04 = O_OpenSeparator
Y[myIO].Y06 = O_Locate
Y[myIO].Y05 = O_OpenStop
END_PROGRAM
```

### Program Logical/Reference/16_pbr2 (IEC) - *PBR2 Bag Remover

#### pbr.var
```iecst
VAR
	LocatedET : TIME;
	Settled : BOOL;
	SettledET : TIME;
	Step3TimedOutET : TIME;
	Step3TimedOut : BOOL;
	SettledAtRemoverET : TIME;
	SettledAtRemover : BOOL;
	STEP : UINT;
	PLS : BOOL;
	LASTSTEP : UINT;
	SeparatorOpened : BOOL;
	SeparatorOpenedET : TIME;
	zzTON_10ms00000 : TON_10ms;
	O_OpenStop : BOOL;
	zzTON_10ms00001 : TON_10ms;
	O_Locate : BOOL;
	O_OpenSeparator : BOOL;
	I_BagReleased : BOOL;
	I_BagAtRemover : BOOL;
	I_BagAtSeparator : BOOL;
	zzTON_10ms00002 : TON_10ms;
	Located : BOOL;
	Step6TimedOutET : TIME;
	Step6TimedOut : BOOL;
	zzTON_10ms00003 : TON_10ms;
	zzTON_10ms00004 : TON_10ms;
	zzTON_10ms00005 : TON_10ms;
	RemoveLocateET : TIME;
	RemoveLocate : BOOL;
	zzTON_10ms00006 : TON_10ms;
	mySeq : UINT;
	TimerAlarm : TON_10ms;
	myIO : UINT;
	myPbr : UINT;
	myZone : INT;
END_VAR
```

### Program Logical/Reference/17_pp3 (IEC) - *PP3 Full bags to PICD 4&5

#### pp.ab
```automation-basic
;--------------------------------------------
;Sequence 0 - XXX0  D[900 + mySeq]
;--------------------------------------------

PROGRAM _INIT
(* init program *)
END_PROGRAM

PROGRAM _CYCLIC

;Inputs
mySeq				= 17	;Sequence number
myIO				= 103
myBag				= 911
myICBufferBag[4]	= 907
myICBufferBag[5]	= 908

myZone	= 1

I_BagAtSep		= X[myIO].X01
I_BagInSep		= X[myIO].X03
I_BagArriveIC[4] = X[174].X03
I_BagArriveIC[5] = X[175].X03

I_InclineBufferClear[4] = (NOT X[174].X02 AND NOT I_BagArriveIC[4] AND NOT Y[174].Y06)
I_InclineBufferClear[5] = (NOT X[175].X02 AND NOT I_BagArriveIC[5] AND NOT Y[175].Y06)

O_OpenSep			= FALSE
O_Select[4]			= FALSE
O_Select[5]			= FALSE

Alarm[mySeq].Name 	= 0
Alarm[mySeq].Bag	= myBag
Alarm[mySeq].Beacon	= TRUE
Alarm[mySeq].Extra	= 0
Alarm[mySeq].Time	= 3000

;Setup Sequence
STEP = D[900 + mySeq]
;Setup Pulse contact
PLS = (STEP <> LASTSTEP)
LASTSTEP = STEP

TON_10ms(I_BagInSep,75,SettledInSep,SettledInSepET)
IF (STEP < 2) THEN
	BagInSep = FALSE
ELSE IF SettledInSep THEN
	BagInSep = TRUE
ENDIF

;Sequence
IF (STEP = 0) THEN
	;Disabled
ENDIF

;step 1 Check destination of bag in buffer
myDest = Bag[myBag].Dst
BagValid = (Bag[myBag].Cat > 0)

TON_10ms(I_BagAtSep,200,SettledAtSep,SettledAtSepET)
TON_10ms(ResetPoints,200,PointsReset,PointsResetET)
IF (STEP = 1) THEN
	IF (myDest > 20) AND (myDest < 24) THEN
		myIC = 4
	ELSE IF	(myDest > 23) AND (myDest < 27) THEN
		myIC = 5
	ELSE
		myIC = 0
	ENDIF
	DestValid = (myIC > 0)
	IF BagValid AND DestValid AND SettledAtSep AND NOT I_BagInSep THEN

		IF (myIC = myPrevIC) AND DestValid THEN
			IF (myDest > 23) THEN
				D[900 + mySeq]  = 4
			ELSE
				D[900 + mySeq]  = 2
			ENDIF
		ELSE
			ResetPoints = TRUE
			IF (myDest > 23) THEN
				O_Select[5] = TRUE
				IF PointsReset THEN
					D[900 + mySeq]  = 4
				ENDIF
			ELSE
				O_Select[4] = TRUE
				IF PointsReset THEN
					D[900 + mySeq]  = 2
				ENDIF
			ENDIF
		ENDIF
	ENDIF
	IF NOT BagValid	AND SettledAtSep THEN
		Alarm[mySeq].Name = almBagDataError
	ELSE IF BagValid AND NOT SettledAtSep THEN
		Alarm[mySeq].Name = almSwitchFault
	ELSE IF NOT DestValid AND SettledAtSep THEN
		Alarm[mySeq].Name = almDestinationNotValid
	ENDIF
ELSE
	ResetPoints = FALSE
ENDIF

;Step 2 Check for space at buffer PIC4
IF (STEP = 2) THEN
	myIC = 4
	myPrevIC = myIC
	DestValid = (myDest > 20) AND (myDest < 24)
	O_Select[myIC] = DestValid
	ReleaseValid = DestValid AND BagValid AND SettledAtSep AND NOT Std.HaltSysZone[myZone]
	InclineClear = ((Bag[myICBufferBag[myIC]].Cat = 0) AND I_InclineBufferClear[myIC])
	IF ReleaseValid AND InclineClear THEN
		D[900 + mySeq] = 3
	ENDIF
	IF NOT BagValid	AND SettledAtSep THEN
		Alarm[mySeq].Name = almBagDataError
	ELSE IF BagValid AND NOT SettledAtSep THEN
		Alarm[mySeq].Name = almSwitchFault
	ELSE IF NOT DestValid AND SettledAtSep THEN
		Alarm[mySeq].Name = almDestinationNotValid
	ENDIF
ENDIF

;Step 3 Release bag to decline 4
IF (STEP = 3) THEN
	myIC = 4
	myPrevIC = myIC
	InclineClear = ((Bag[myICBufferBag[myIC]].Cat = 0) AND I_InclineBufferClear[myIC])
	DestValid = (myDest > 20) AND (myDest < 24)
	O_Select[myIC] = DestValid
	O_OpenSep = InclineClear AND DestValid AND BagValid AND NOT BagInSep
	IF I_BagArriveIC[myIC] THEN
		Bag[myICBufferBag[myIC]] = Bag[myBag]
		Bag[myBag] = Bag[0]
		D[900 + mySeq] = 1
	ENDIF
	IF NOT BagValid	AND SettledAtSep THEN
		Alarm[mySeq].Name = almBagDataError
	ELSE IF BagValid AND NOT SettledAtSep THEN
		Alarm[mySeq].Name = almSwitchFault
	ELSE IF NOT DestValid AND SettledAtSep THEN
		Alarm[mySeq].Name = almDestinationNotValid
	ENDIF
ENDIF

;Step 4 Check for space at buffer PIC5
IF (STEP = 4) THEN
	myIC = 5
	myPrevIC = myIC
	DestValid = (myDest > 23) AND (myDest < 27)
	O_Select[myIC] = DestValid
	ReleaseValid = DestValid AND BagValid AND SettledAtSep AND NOT Std.HaltSysZone[myZone]
	InclineClear = ((Bag[myICBufferBag[myIC]].Cat = 0) AND I_InclineBufferClear[myIC])
	IF ReleaseValid AND InclineClear THEN
		D[900 + mySeq] = 5
	ENDIF
	IF NOT BagValid	AND SettledAtSep THEN
		Alarm[mySeq].Name = almBagDataError
	ELSE IF BagValid AND NOT SettledAtSep THEN
		Alarm[mySeq].Name = almSwitchFault
	ELSE IF NOT DestValid AND SettledAtSep THEN
		Alarm[mySeq].Name = almDestinationNotValid
	ENDIF
ENDIF

;Step 5 Release bag to decline 5
IF (STEP = 5) THEN
	myIC = 5
	myPrevIC = myIC
	InclineClear = ((Bag[myICBufferBag[myIC]].Cat = 0) AND I_InclineBufferClear[myIC])
	DestValid = (myDest > 23) AND (myDest < 27)
	O_Select[myIC] = DestValid
	O_OpenSep = InclineClear AND DestValid AND BagValid AND NOT BagInSep
	IF I_BagArriveIC[myIC] THEN
		Bag[myICBufferBag[myIC]] = Bag[myBag]
		Bag[myBag] = Bag[0]
		D[900 + mySeq] = 1
	ENDIF
	IF NOT BagValid	AND SettledAtSep THEN
		Alarm[mySeq].Name = almBagDataError
	ELSE IF BagValid AND NOT SettledAtSep THEN
		Alarm[mySeq].Name = almSwitchFault
	ELSE IF NOT DestValid AND SettledAtSep THEN
		Alarm[mySeq].Name = almDestinationNotValid
	ENDIF
ENDIF

;-----------------------------------
;PLC Outputs - adjust to suit system
;-----------------------------------

Y[myIO].Y05 = O_OpenSep
Y[myIO].Y07 = O_Select[4]
Y[myIO].Y08 = O_Select[5]

;Alarms
TimerAlarm.IN 		= NOT PLS AND (Alarm[mySeq].Name > 0)
TimerAlarm.PT 		= Alarm[mySeq].Time
TimerAlarm FUB TON_10ms()
Alarm[mySeq].On 	= TimerAlarm.Q
Alarm[mySeq].ET 	= TimerAlarm.ET
Alarm[mySeq].Zone 	= myZone
END_PROGRAM
```

### Program Logical/Reference/18_pp4 (IEC) - *PP4 Full bag from PID4

#### pp.var
```iecst
VAR
	BagReleased : BOOL;
	BagValid : BOOL;
	DestValid : BOOL;
	I_BagAtSep : BOOL;
	I_BagInSep : BOOL;
END_VAR
VAR RETAIN
	LASTSTEP : UINT;
END_VAR
VAR
	LineValid : ARRAY[0..2] OF BOOL;
	myBag : UINT;
	myDest : USINT;
	myIO : UINT;
	myIO2 : UINT;
	myPrevSelLine : USINT;
	myRelLastBag : ARRAY[0..2] OF UINT;
	myRelLine : ARRAY[0..2] OF UINT;
	mySelLine : USINT;
	mySeq : UINT;
	myZone : INT;
	O_OpenSep : BOOL;
	O_Select : ARRAY[0..2] OF BOOL;
END_VAR
VAR RETAIN
	PLS : BOOL;
END_VAR
VAR
	PointsReset : BOOL;
	PointsResetET : UDINT;
	ResetPoints : BOOL;
	SettledAtSep : BOOL;
	SettledAtSepET : UDINT;
END_VAR
VAR RETAIN
	STEP : UINT;
END_VAR
VAR
	TimerAlarm : TON_10ms;
	SettledInSep : BOOL;
	SettledInSepET : UDINT;
	BagInSep : BOOL;
END_VAR
```

#### pp.ab
```automation-basic
;--------------------------------------------
;Sequence 0 - XXX0  D[900 + mySeq]
;--------------------------------------------

PROGRAM _INIT
(* init program *)
END_PROGRAM

PROGRAM _CYCLIC

;Inputs
mySeq				= 18	;Sequence number
myIO				= 104
myIO2				= 124
myBag				= 935
myRelLine[1]		= 72
myRelLine[2]		= 76
myRelLastBag[1]		= Line[myRelLine[1]].LastBag
myRelLastBag[2]		= Line[myRelLine[2]].LastBag

myZone	= 0

I_BagAtSep			= X[myIO2].X01
I_BagInSep			= X[myIO2].X03

O_OpenSep			= FALSE
O_Select[1]			= FALSE
O_Select[2]			= FALSE

Alarm[mySeq].Name 	= 0
Alarm[mySeq].Bag	= 0
Alarm[mySeq].Beacon	= TRUE
Alarm[mySeq].Extra	= 0
Alarm[mySeq].Time	= 3000

;Setup Sequence
STEP = D[900 + mySeq]
;Setup Pulse contact
PLS = (STEP <> LASTSTEP)
LASTSTEP = STEP

;Sequence
IF (STEP = 0) THEN
	;Disabled
ENDIF
TON_10ms(I_BagInSep,75,SettledInSep,SettledInSepET)
IF (STEP < 2) THEN
	BagInSep = FALSE
ELSE IF SettledInSep THEN
	BagInSep = TRUE
ENDIF

myDest = Bag[myBag].Dst
BagValid = (Bag[myBag].Cat > 0)
LineValid[1] = (Line[myRelLine[1]].Clear AND NOT Line[myRelLine[1]].TripFault) ; Line clear checks bag data and long trip made for 3 secs.
LineValid[2] = (Line[myRelLine[2]].Clear AND NOT Line[myRelLine[2]].TripFault)

TON_10ms(I_BagAtSep,100,SettledAtSep,SettledAtSepET)
TON_10ms(ResetPoints,100,PointsReset,PointsResetET)
IF (STEP = 1) THEN
	IF (myDest = 21) THEN
		mySelLine = 1
	ELSE IF	(myDest > 21) AND (myDest < 24) THEN
		mySelLine = 2
	ELSE
		mySelLine = 0
	ENDIF
	DestValid = (mySelLine > 0)
	IF BagValid AND DestValid AND SettledAtSep AND NOT I_BagInSep AND NOT Std.HaltSysZone[myZone] THEN
		IF (mySelLine = myPrevSelLine) AND DestValid THEN
			IF LineValid[mySelLine] THEN
				D[900 + mySeq] = (mySelLine + 1)
			ENDIF
		ELSE
			ResetPoints = TRUE
			O_Select[mySelLine] = TRUE
			IF PointsReset AND LineValid[mySelLine] THEN
				D[900 + mySeq] = (mySelLine + 1)
			ENDIF
		ENDIF
	ENDIF
	IF NOT BagValid	AND SettledAtSep THEN
		Alarm[mySeq].Name = almBagDataError
	ELSE IF BagValid AND NOT SettledAtSep THEN
		Alarm[mySeq].Name = almSwitchFault
	ELSE IF NOT DestValid AND SettledAtSep THEN
		Alarm[mySeq].Name = almDestinationNotValid
	ENDIF
ELSE
	ResetPoints = FALSE
ENDIF

;Step 2 Release bag to PUP 1
IF (STEP = 2) THEN
	mySelLine = 1
	myPrevSelLine = mySelLine
	DestValid = (myDest = 21)
	O_Select[mySelLine] = DestValid
	O_OpenSep = DestValid AND BagValid AND LineValid[mySelLine] AND NOT BagInSep
	IF Line[myRelLine[mySelLine]].Trip THEN
		Bag[myRelLastBag[mySelLine]] = Bag[myBag]
		Bag[myBag] = Bag[0]
		D[900 + mySeq] = 1
	ENDIF
	IF NOT BagValid	AND SettledAtSep THEN
		Alarm[mySeq].Name = almBagDataError
	ELSE IF BagValid AND NOT SettledAtSep THEN
		Alarm[mySeq].Name = almSwitchFault
	ELSE IF NOT DestValid AND SettledAtSep THEN
		Alarm[mySeq].Name = almDestinationNotValid
	ENDIF
ENDIF

;Step 3 Release bag to PUP 2,3
IF (STEP = 3) THEN
	mySelLine = 2
	myPrevSelLine = mySelLine
	DestValid = ((myDest = 22) OR (myDest = 23))
	O_Select[mySelLine] = DestValid
	O_OpenSep = DestValid AND BagValid AND LineValid[mySelLine] AND NOT BagInSep
	IF Line[myRelLine[mySelLine]].Trip THEN
		Bag[myRelLastBag[mySelLine]] = Bag[myBag]
		Bag[myBag] = Bag[0]
		D[900 + mySeq] = 1
	ENDIF
	IF NOT BagValid	AND SettledAtSep THEN
		Alarm[mySeq].Name = almBagDataError
	ELSE IF BagValid AND NOT SettledAtSep THEN
		Alarm[mySeq].Name = almSwitchFault
	ELSE IF NOT DestValid AND SettledAtSep THEN
		Alarm[mySeq].Name = almDestinationNotValid
	ENDIF
ENDIF

;-----------------------------------
;PLC Outputs - adjust to suit system
;-----------------------------------

Y[myIO].Y07 	= O_Select[2]
Y[myIO].Y08 	= O_Select[1]
Y[myIO2].Y05 	= O_OpenSep

;Alarms
TimerAlarm.IN 		= NOT PLS AND (Alarm[mySeq].Name > 0)
TimerAlarm.PT 		= Alarm[mySeq].Time
TimerAlarm FUB TON_10ms()
Alarm[mySeq].On 	= TimerAlarm.Q
Alarm[mySeq].ET 	= TimerAlarm.ET
Alarm[mySeq].Zone 	= myZone
END_PROGRAM
```

### Program Logical/Reference/20_pp6 (IEC) - *PP6 Empty trolleys feeding PICU7

#### pp.ab
```automation-basic
;--------------------------------------------
;Sequence 0 - XXX0  D[900 + mySeq]
;--------------------------------------------

PROGRAM _INIT
(* init program *)
END_PROGRAM

PROGRAM _CYCLIC

;Inputs
mySeq				= 20	;Sequence number
myIO				= 106
myZone				= 0

TrolleyBatchSize 	= 1

I_BagAtSep[1]			= RequestRel.IC[6]	;X[myIO].X01
I_BagAtSep[2]			= X[myIO].X02
I_BagInSep[2]			= X[myIO].X04
I_LineFull				= X[myIO].X03
I_BufferLineFull[1]		= X[346].X08
I_BufferLineFull[2]		= X[345].X08

O_OpenSep[1]			= FALSE
O_OpenSep[2]			= FALSE
O_Select[1]				= FALSE
O_Select[2]				= FALSE
EnableRel.IC[6]			= FALSE

Alarm[mySeq].Name 	= 0
Alarm[mySeq].Bag	= 10000 + mySeq
Alarm[mySeq].Beacon	= TRUE
Alarm[mySeq].Extra	= 0
Alarm[mySeq].Time	= 3000

;Setup Sequence
STEP = D[900 + mySeq]
;Setup Pulse contact
PLS = (STEP <> LASTSTEP)
LASTSTEP = STEP

;Keep trolley counts inrange
LOOP n = 1 TO 2 DO
	IF (TrolleyCount[n] >$FFFE) THEN
		TrolleyCount[n] = $FFFE
	ENDIF
ENDLOOP

;Sequence
IF (STEP = 0) THEN
	;Disabled
ENDIF

;Step 1 Decide where to take trolley from
TON_10ms(I_BagAtSep[1],250,SettledAtSep[1],SettledAtSepET[1])
TON_10ms(I_BagAtSep[2],250,SettledAtSep[2],SettledAtSepET[2])
TON_10ms(I_BufferLineFull[1],400,BufferFull[1],BufferFullET[1])
TON_10ms(I_BufferLineFull[2],400,BufferFull[2],BufferFullET[2])
TON_10ms(Reset,200,ResetPoints,ResetPointsET)
IF (STEP = 1) THEN
		;Force line choice if line is full
	IF NOT Reset THEN
		IF BufferFull[1] AND NOT BufferFull[2] THEN
			myLine = 1
		ELSE IF BufferFull[2] AND NOT BufferFull[1] THEN
			myLine = 2
		ENDIF
	ENDIF
	IF (myLine = 0) OR (myLine > 2) THEN
		myLine = 1
	ENDIF

	IF (SettledAtSep[myLine] AND (TrolleyCount[myLine] < TrolleyBatchSize) AND NOT I_LineFull AND NOT Reset AND NOT Std.HaltSysZone[myZone]) THEN
		IF (myLine = myPrevLine) THEN
			D[900 +  mySeq] = (myLine + 1)
		ELSE
			Reset = TRUE
		ENDIF
	ELSE IF Reset THEN
		O_Select[myLine] = TRUE
		IF ResetPoints THEN
			myPrevLine = myLine
			D[900 +  mySeq] = (myLine + 1)
		ENDIF
	ELSE IF (TrolleyCount[myLine] >= TrolleyBatchSize) OR NOT I_BagAtSep[myLine] THEN
		TrolleyCount[myLine] = 0
		INC myLine
	ENDIF
ELSE
	Reset = FALSE
ENDIF
;Step 2 Select Line 1
IF (STEP = 2) THEN
	myLine = 1
	O_Select[myLine] = TRUE
	O_OpenSep[myLine] = TRUE
	IF I_LineFull THEN
		INC TrolleyCount[myLine]
		D[900 + mySeq] = 1
	ENDIF
	Alarm[mySeq].Name = almBagNotReleased
ENDIF

;Step 3 Select Line 2
TON_10ms(I_BagInSep[2],200,SettledInSep[2],SettledInSepET[2])
IF (STEP = 3) THEN
	myLine = 2
	IF SettledInSep[myLine] THEN
		BagInSep = TRUE
	ENDIF
	O_Select[myLine] = TRUE
	O_OpenSep[myLine] = NOT BagInSep
	IF I_LineFull THEN
		INC TrolleyCount[myLine]
		D[900 + mySeq] = 1
	ENDIF
	Alarm[mySeq].Name = almBagNotReleased
ELSE
	BagInSep = FALSE
ENDIF

;-----------------------------------
;PLC Outputs - adjust to suit system
;-----------------------------------

;Y[myIO].Y05 = O_OpenSep[1]
EnableRel.IC[6]	= O_OpenSep[1]
Y[myIO].Y06 = O_OpenSep[2]
Y[myIO].Y07 = O_Select[1]
Y[myIO].Y08 = O_Select[2]

;Alarms
TimerAlarm.IN 		= NOT PLS AND (Alarm[mySeq].Name > 0)
TimerAlarm.PT 		= Alarm[mySeq].Time
TimerAlarm FUB TON_10ms()
Alarm[mySeq].On 	= TimerAlarm.Q
Alarm[mySeq].ET 	= TimerAlarm.ET
Alarm[mySeq].Zone 	= myZone
END_PROGRAM
```

### Program Logical/Reference/22_pp8 (IEC) - *PP8 Full bag from PID5

#### pp.ab
```automation-basic
;--------------------------------------------
;Sequence 0 - XXX0  D[900 + mySeq]
;--------------------------------------------

PROGRAM _INIT
(* init program *)
END_PROGRAM

PROGRAM _CYCLIC

;Inputs
mySeq				= 22	;Sequence number
myIO				= 108
myIO2				= 128
myBag				= 940
myRelLine[1]		= 71
myRelLine[2]		= 75
myRelLastBag[1]		= Line[myRelLine[1]].LastBag
myRelLastBag[2]		= Line[myRelLine[2]].LastBag

myZone	= 0

I_BagAtSep			= X[myIO2].X01
I_BagInSep			= X[myIO2].X03

O_OpenSep			= FALSE
O_Select[1]			= FALSE
O_Select[2]			= FALSE

Alarm[mySeq].Name 	= 0
Alarm[mySeq].Bag	= 0
Alarm[mySeq].Beacon	= TRUE
Alarm[mySeq].Extra	= 0
Alarm[mySeq].Time	= 3000

;Setup Sequence
STEP = D[900 + mySeq]
;Setup Pulse contact
PLS = (STEP <> LASTSTEP)
LASTSTEP = STEP

;Sequence
IF (STEP = 0) THEN
	;Disabled
ENDIF
TON_10ms(I_BagInSep,75,SettledInSep,SettledInSepET)
IF (STEP < 2) THEN
	BagInSep = FALSE
ELSE IF SettledInSep THEN
	BagInSep = TRUE
ENDIF

myDest = Bag[myBag].Dst
BagValid = (Bag[myBag].Cat > 0)
LineValid[1] = (Line[myRelLine[1]].Clear AND NOT Line[myRelLine[1]].TripFault) ; Line clear checks bag data and long trip made for 3 secs.
LineValid[2] = (Line[myRelLine[2]].Clear AND NOT Line[myRelLine[2]].TripFault)

TON_10ms(I_BagAtSep,75,SettledAtSep,SettledAtSepET)
TON_10ms(ResetPoints,100,PointsReset,PointsResetET)
IF (STEP = 1) THEN
	IF (myDest = 24) THEN
		mySelLine = 1
	ELSE IF	(myDest > 24) AND (myDest < 27) THEN
		mySelLine = 2
	ELSE
		mySelLine = 0
	ENDIF
	DestValid = (mySelLine > 0)
	IF BagValid AND DestValid AND SettledAtSep AND NOT I_BagInSep AND NOT Std.HaltSysZone[myZone] THEN
		IF (mySelLine = myPrevSelLine) AND DestValid THEN
			IF LineValid[mySelLine] THEN
				D[900 + mySeq] = (mySelLine + 1)
			ENDIF
		ELSE
			ResetPoints = TRUE
			O_Select[mySelLine] = TRUE
			IF PointsReset AND LineValid[mySelLine] THEN
				D[900 + mySeq] = (mySelLine + 1)
			ENDIF
		ENDIF
	ENDIF
	IF NOT BagValid	AND SettledAtSep THEN
		Alarm[mySeq].Name = almBagDataError
	ELSE IF BagValid AND NOT SettledAtSep THEN
		Alarm[mySeq].Name = almSwitchFault
	ELSE IF NOT DestValid AND SettledAtSep THEN
		Alarm[mySeq].Name = almDestinationNotValid
	ENDIF
ELSE
	ResetPoints = FALSE
ENDIF

;Step 2 Release bag to PUP 1
IF (STEP = 2) THEN
	mySelLine = 1
	myPrevSelLine = mySelLine
	DestValid = (myDest = 24)
	O_Select[mySelLine] = DestValid
	O_OpenSep = DestValid AND BagValid AND LineValid[mySelLine] AND NOT BagInSep
	IF Line[myRelLine[mySelLine]].Trip THEN
		Bag[myRelLastBag[mySelLine]] = Bag[myBag]
		Bag[myBag] = Bag[0]
		D[900 + mySeq] = 1
	ENDIF
	IF NOT BagValid	AND SettledAtSep THEN
		Alarm[mySeq].Name = almBagDataError
	ELSE IF BagValid AND NOT SettledAtSep THEN
		Alarm[mySeq].Name = almSwitchFault
	ELSE IF NOT DestValid AND SettledAtSep THEN
		Alarm[mySeq].Name = almDestinationNotValid
	ENDIF
ENDIF

;Step 3 Release bag to PUP 2,3
IF (STEP = 3) THEN
	mySelLine = 2
	myPrevSelLine = mySelLine
	DestValid = ((myDest = 25) OR (myDest = 26))
	O_Select[mySelLine] = DestValid
	O_OpenSep = DestValid AND BagValid AND LineValid[mySelLine] AND NOT BagInSep
	IF Line[myRelLine[mySelLine]].Trip THEN
		Bag[myRelLastBag[mySelLine]] = Bag[myBag]
		Bag[myBag] = Bag[0]
		D[900 + mySeq] = 1
	ENDIF
	IF NOT BagValid	AND SettledAtSep THEN
		Alarm[mySeq].Name = almBagDataError
	ELSE IF BagValid AND NOT SettledAtSep THEN
		Alarm[mySeq].Name = almSwitchFault
	ELSE IF NOT DestValid AND SettledAtSep THEN
		Alarm[mySeq].Name = almDestinationNotValid
	ENDIF
ENDIF

;-----------------------------------
;PLC Outputs - adjust to suit system
;-----------------------------------

Y[myIO].Y07 	= O_Select[1]
Y[myIO].Y08 	= O_Select[2]
Y[myIO2].Y05 	= O_OpenSep

;Alarms
TimerAlarm.IN 		= NOT PLS AND (Alarm[mySeq].Name > 0)
TimerAlarm.PT 		= Alarm[mySeq].Time
TimerAlarm FUB TON_10ms()
Alarm[mySeq].On 	= TimerAlarm.Q
Alarm[mySeq].ET 	= TimerAlarm.ET
Alarm[mySeq].Zone 	= myZone
END_PROGRAM
```

### Program Logical/Reference/23_pp9 (IEC) - *PP9 Full bags to PUP 5&6

#### pp.var
```iecst
VAR
	BagReleased : BOOL;
	BagValid : BOOL;
	DestValid : BOOL;
	I_BagAtSep : BOOL;
	I_BagReleased : BOOL;
END_VAR
VAR RETAIN
	LASTSTEP : UINT;
END_VAR
VAR
	myBag : UINT;
	myDest : USINT;
	myIC : USINT;
	myIO : UINT;
END_VAR
VAR RETAIN
	myPrevSelLine : USINT;
END_VAR
VAR
	myPUP : ARRAY[0..2] OF USINT;
	myRelDest : ARRAY[0..2] OF USINT;
	mySelLine : USINT;
	mySeq : UINT;
	O_OpenSep : BOOL;
	O_Select : ARRAY[0..9] OF BOOL;
END_VAR
VAR RETAIN
	PLS : BOOL;
END_VAR
VAR
	PointsReset : BOOL;
	PointsResetET : UDINT;
	ResetPoints : BOOL;
	SettledAtSep : BOOL;
	SettledAtSepET : UDINT;
END_VAR
VAR RETAIN
	STEP : UINT;
END_VAR
VAR
	TimerAlarm : TON_10ms;
	I_BagArrive : ARRAY[0..2] OF BOOL;
	myOutBag : ARRAY[0..2] OF UINT;
	PUPClear : ARRAY[0..2] OF BOOL;
	myZone : INT;
	I_BagInSep : BOOL;
	SettledInSep : BOOL;
	SettledInSepET : UDINT;
	BagInSep : BOOL;
	ReleaseValid : BOOL;
	AutoDestChange : BOOL;
END_VAR
```

### Program Logical/Reference/26_pp12 (IEC) - *PP12 Empty trolleys from PUP 1-6

#### pp.var
```iecst
VAR RETAIN
	LASTSTEP : UINT;
	PLS : BOOL;
	STEP : UINT;
END_VAR
VAR
	TimerAlarm : TON_10ms;
	mySeq : UINT;
	myIO : UINT;
	I_BagAtSep : ARRAY[0..2] OF BOOL;
	I_LineFull : BOOL;
	O_OpenSep : ARRAY[0..2] OF BOOL;
	O_Select : ARRAY[0..2] OF BOOL;
	SettledAtSep : ARRAY[0..2] OF BOOL;
	SettledAtSepET : ARRAY[0..2] OF UDINT;
	myLine : USINT;
	TrolleyCount : ARRAY[0..2] OF UINT;
	TrolleyBatchSize : UINT;
	n : UINT;
	I_BufferLineFull : ARRAY[0..2] OF BOOL;
	BufferFull : ARRAY[0..2] OF BOOL;
	BufferFullET : ARRAY[0..2] OF UDINT;
	Reset : BOOL;
	ResetPoints : BOOL;
	ResetPointsET : UDINT;
END_VAR
VAR RETAIN
	myPrevLine : UINT;
END_VAR
VAR
	myZone : INT;
	BatchRecieved : BOOL;
	CloseStop : BOOL;
	CloseStopET : UDINT;
	WholeBatchRecieved : BOOL;
	WholeBatchRecievedET : UDINT;
END_VAR
```

### Program Logical/Reference/27_pp13 (IEC) - *PP13 Empty trolleys to PICD13 + PP14

#### pp.var
```iecst
VAR RETAIN
	LASTSTEP : UINT;
	PLS : BOOL;
	STEP : UINT;
END_VAR
VAR
	TimerAlarm : TON_10ms;
	mySeq : UINT;
	myIO : UINT;
	I_BagAtBuffer : BOOL;
	I_BagAtSep : BOOL;
	I_LineFull : ARRAY[0..2] OF BOOL;
	O_OpenSep : BOOL;
	O_Select : ARRAY[0..2] OF BOOL;
	n : UINT;
	TrolleyCount : ARRAY[0..2] OF UINT;
	SettledAtSep : BOOL;
	SettledAtSepET : UDINT;
	Reset : BOOL;
	ResetPoints : BOOL;
	ResetPointsET : UDINT;
	myLine : UINT;
	TrolleyBatchSize : UINT;
	myPrevLine : UINT;
	I_BufferLineEmpty : ARRAY[0..2] OF BOOL;
	BufferEmpty : ARRAY[0..2] OF BOOL;
	BufferEmptyET : ARRAY[0..2] OF UDINT;
	myZone : INT;
	OpenStopTime : UDINT;
	OpenStop : BOOL;
	OpenStopET : UDINT;
	BagsArrived : BOOL;
	BagsReleased : BOOL;
	BagsReleasedET : UDINT;
END_VAR
```

### Program Logical/Reference/28_pp14 (IEC) - *PP14 Empty trolleys to PICD14+ PICD15

#### pp.ab
```automation-basic
;--------------------------------------------
;Sequence 0 - XXX0  D[900 + mySeq]
;--------------------------------------------

PROGRAM _INIT
(* init program *)
END_PROGRAM

PROGRAM _CYCLIC

;Inputs
mySeq				= 28	;Sequence number
myIO				= 114
myZone				= 3

I_BagAtSep			= X[myIO].X01
I_LineFull[1]		= X[myIO].X03
I_LineFull[2]		= X[myIO].X04
I_BufferLineEmpty[1] = 	(NOT X[184].X03 AND NOT Y[184].Y06)
I_BufferLineEmpty[2] = 	(NOT X[185].X03 AND NOT Y[185].Y06)

TrolleyBatchSize	= 3

O_OpenSep			= FALSE
O_Select[1]			= FALSE
O_Select[2]			= FALSE

Alarm[mySeq].Name 	= 0
Alarm[mySeq].Bag	= 10000 + mySeq
Alarm[mySeq].Beacon	= TRUE
Alarm[mySeq].Extra	= 0
Alarm[mySeq].Time	= 3000
IF OpenStopTime = 0 THEN
	OpenStopTime 		= 100
ENDIF

;Setup Sequence
STEP = D[900 + mySeq]
;Setup Pulse contact
PLS = (STEP <> LASTSTEP)
LASTSTEP = STEP

;Sequence
IF (STEP = 0) THEN
	;Disabled
ENDIF

;Step 1 Decide where to send trolley
TON_10ms(I_BagAtSep,250,SettledAtSep,SettledAtSepET)
TON_10ms(I_BufferLineEmpty[1],200,BufferEmpty[1],BufferEmptyET[1])
TON_10ms(I_BufferLineEmpty[2],200,BufferEmpty[2],BufferEmptyET[2])
TON_10ms((STEP = 1),200,ResetPoints,ResetPointsET)
IF (STEP = 1) THEN
	BagsArrived = FALSE
	IF (SettledAtSep AND NOT Std.HaltSysZone[myZone]) THEN
		IF (myLine < 2) THEN
			INC myLine
		ELSE
			myLine = 1
		ENDIF

		IF NOT I_LineFull[myLine]  THEN
			D[900 +  mySeq] = (myLine + 1)
		ENDIF
	ENDIF
ENDIF

TON_10ms((STEP = 2) OR (STEP = 3),OpenStopTime,OpenStop,OpenStopET)
TON_10ms(BagsArrived,OpenStopTime + 100,BagsReleased,BagsReleasedET)
;Step 2 Select Line 1
IF (STEP = 2) THEN
	myLine = 1
	OpenStopTime = 100
	O_Select[myLine] = TRUE
	O_OpenSep = NOT OpenStop
	IF I_LineFull[myLine] THEN
		BagsArrived = TRUE
	ENDIF
	IF BagsReleased THEN
		D[900 + mySeq] = 1
	ENDIF
	Alarm[mySeq].Name = almBagNotReleased
ENDIF

;Step 3 Select Line 2
IF (STEP = 3) THEN
	myLine = 2
	OpenStopTime = 200
	O_Select[myLine] = TRUE
	O_OpenSep = NOT OpenStop
	IF I_LineFull[myLine] THEN
		BagsArrived = TRUE
	ENDIF
	IF BagsReleased THEN
		D[900 + mySeq] = 1
	ENDIF
	Alarm[mySeq].Name = almBagNotReleased
ENDIF

;-----------------------------------
;PLC Outputs - adjust to suit system
;-----------------------------------

Y[myIO].Y05 = O_OpenSep
Y[myIO].Y07 = O_Select[1]
Y[myIO].Y08 = O_Select[2]

;Alarms
TimerAlarm.IN 		= NOT PLS AND (Alarm[mySeq].Name > 0)
TimerAlarm.PT 		= Alarm[mySeq].Time
TimerAlarm FUB TON_10ms()
Alarm[mySeq].On 	= TimerAlarm.Q
Alarm[mySeq].ET 	= TimerAlarm.ET
Alarm[mySeq].Zone 	= myZone
END_PROGRAM
```

### Program Logical/Reference/30_picu1 (IEC) - *PICU1 Incline Up Full bags

#### picu.ab
```automation-basic
PROGRAM _CYCLIC

;Sequence 24 - Primary Incline Conveyor 1 D[900 + mySeq]

;Note - Not a real sequence and not shown

;-----------------------------------------
;Revision 1.00 17/04/2007 D.J. First Issue
;-----------------------------------------

mySeq = 30
myIO = 171
myX20IO	= 23
myBufferBag = 831
myRelLine	= 66
myLine = 81 ; Line used to track bags
myZone	= 4

myLastBag = Line[myLine].LastBag
myFirstBag = Line[myLine].FirstBag
myRelBag = Line[myRelLine].LastBag

I_PaddleInPosition		= X[myIO].X01
I_BagReleasedSep		= X[myIO].X02
I_BagAtSep              = X[myIO].X03
I_ArriveIncline			= X[myIO].X04

O_RunMotor 				= FALSE
O_OpenSeparator			= FALSE

Alarm[mySeq].Name 	= 0
Alarm[mySeq].Bag	= myFirstBag
Alarm[mySeq].Beacon	= TRUE
Alarm[mySeq].Extra	= 0
Alarm[mySeq].Time	= 3000

;Setup Sequence
;-----------------------
STEP = D[900 + mySeq]
;Setup Pulse contact
PLS = (STEP <> LASTSTEP)
LASTSTEP = STEP

;If no bags on the buffers then stop the motor
NoBags = (Bag[myBufferBag].Cat = 0) AND (Bag[myFirstBag].Cat = 0)
TON_10ms(NoBags,10,StopIncline,StopInclineET)

O_RunMotor = (Line[myRelLine].Clear AND NOT Line[myRelLine].TripFault AND NOT StopIncline AND NOT Std.HaltSysZone[myZone] AND (STEP <> 2) AND (STEP <> 0))
IF (STEP = 0) THEN

ENDIF

;Run Incline until paddle in position
TON_10ms(I_BagAtSep,250,SettledInSep,SettledInSepET)
TON_10ms((Bag[myBufferBag].Cat > 0) AND NOT Std.HaltSysZone[myZone],300,SettledAtSep,SettledAtSepET)
IF (STEP = 1) THEN
	IF (I_PaddleInPosition AND O_RunMotor AND SettledAtSep AND (Bag[myLastBag].Cat = 0) AND (Bag[myBufferBag].Cat > 0)) THEN
		D[900 + mySeq] = 2
	ENDIF
ENDIF

;Release Bag into incline
IF (STEP = 2) THEN
	IF SettledInSep THEN
		BagArrived = TRUE
	ENDIF
	O_OpenSeparator	= (Bag[myLastBag].Cat = 0) AND NOT BagArrived

	IF I_ArriveIncline THEN
		IF ((Bag[myBufferBag].Cat > 0) AND (Bag[myLastBag].Cat = 0)) THEN
			Bag[myLastBag] = Bag[myBufferBag]
			Bag[myBufferBag] = Bag[0]
		ENDIF
		D[900 + mySeq] = 3
	ENDIF
	IF (Bag[myLastBag].Cat > 0) THEN
		Alarm[mySeq].Name = almBagDataError
		Alarm[mySeq].Time = 0
		Alarm[mySeq].Bag = myLastBag
	ELSE IF (Bag[myBufferBag].Cat > 0) AND NOT I_BagAtSep THEN
		Alarm[mySeq].Name = almSwitchFault
		Alarm[mySeq].Bag = myBufferBag
	ELSE
		Alarm[mySeq].Name = almBagNotReleased
		Alarm[mySeq].Bag = myBufferBag
	ENDIF
ELSE
	BagArrived = FALSE
ENDIF

;Check not stpped on paddle
IF (STEP = 3) THEN
	IF NOT I_PaddleInPosition THEN
		D[900 + mySeq] = 1
	ENDIF
ENDIF

;Move data from incline..
IF Line[myRelLine].Trip AND (Bag[myFirstBag].Cat > 0) AND (Bag[myRelBag].Cat = 0)  THEN ; Trip includes debounce
	Bag[myRelBag] = Bag[myFirstBag]
	Bag[myFirstBag] = Bag[0]
ENDIF

;Alarms
TimerAlarm.IN 		= NOT PLS AND (Alarm[mySeq].Name > 0)
TimerAlarm.PT 		= Alarm[mySeq].Time
TimerAlarm FUB TON_10ms()
Alarm[mySeq].On 	= TimerAlarm.Q
Alarm[mySeq].ET 	= TimerAlarm.ET
Alarm[mySeq].Zone 	= myZone
Y[myX20IO].Y01 	= O_RunMotor
Y[myIO].Y06 	= O_OpenSeparator
END_PROGRAM
```

### Program Logical/Reference/31_picu13 (IEC) - *PICU2 Incline Up Full bags
